C01791=1027.704,285.266,-126.131,170.638,46.717,159.004
C01792=1027.711,285.514,-126.162,170.643,46.715,159.005
C01793=1027.718,285.761,-126.193,170.647,46.714,159.005
C01794=1027.724,286.009,-126.225,170.651,46.713,159.005
C01795=1027.731,286.257,-126.256,170.655,46.712,159.005
C01796=1027.738,286.505,-126.288,170.660,46.711,159.006
C01797=1027.744,286.753,-126.319,170.664,46.710,159.006
C01798=1027.751,287.001,-126.351,170.668,46.709,159.006
C01799=1027.758,287.249,-126.382,170.673,46.708,159.006
C01800=1027.764,287.497,-126.414,170.678,46.706,159.007
C01801=1027.771,287.744,-126.446,170.682,46.705,159.007
C01802=1027.778,287.992,-126.478,170.686,46.704,159.007
C01803=1027.784,288.240,-126.509,170.690,46.703,159.008
C01804=1027.791,288.488,-126.541,170.695,46.702,159.008
C01805=1027.798,288.736,-126.572,170.699,46.701,159.008
C01806=1027.805,288.983,-126.604,170.703,46.700,159.008
C01807=1027.811,289.232,-126.636,170.708,46.699,159.009
C01808=1027.818,289.479,-126.668,170.712,46.698,159.009
C01809=1027.824,289.727,-126.699,170.716,46.697,159.009
C01810=1027.832,289.975,-126.732,170.720,46.696,159.010
C01811=1027.839,290.223,-126.763,170.725,46.695,159.010
C01812=1027.845,290.471,-126.795,170.730,46.694,159.010
C01813=1027.852,290.719,-126.827,170.734,46.693,159.011
C01814=1027.858,290.967,-126.859,170.739,46.692,159.011
C01815=1027.865,291.215,-126.890,170.743,46.691,159.011
C01816=1027.872,291.462,-126.922,170.747,46.690,159.011
C01817=1027.883,291.868,-126.974,170.754,46.689,159.012
C01818=1027.894,292.273,-127.027,170.761,46.687,159.012
C01819=1027.906,292.679,-127.079,170.769,46.685,159.013
C01820=1027.917,293.084,-127.132,170.776,46.684,159.014
C01821=1027.923,293.332,-127.163,170.781,46.683,159.014
C01822=1027.930,293.579,-127.196,170.785,46.682,159.014
C01823=1027.937,293.828,-127.228,170.789,46.681,159.015
C01824=1027.944,294.075,-127.260,170.794,46.680,159.015
C01825=1027.950,294.323,-127.293,170.798,46.679,159.015
C01826=1027.957,294.571,-127.324,170.803,46.679,159.016
C01827=1027.963,294.818,-127.357,170.807,46.678,159.016
C01828=1027.970,295.066,-127.390,170.812,46.677,159.016
C01829=1027.977,295.314,-127.422,170.816,46.676,159.017
C01830=1027.983,295.562,-127.454,170.821,46.675,159.017
C01831=1027.990,295.810,-127.487,170.826,46.675,159.018
C01832=1027.997,296.058,-127.519,170.830,46.674,159.018
C01833=1028.003,296.305,-127.552,170.834,46.673,159.018
C01834=1028.010,296.553,-127.585,170.838,46.672,159.019
C01835=1028.017,296.800,-127.617,170.844,46.671,159.019
C01836=1028.024,297.048,-127.650,170.848,46.671,159.019
C01837=1028.030,297.297,-127.682,170.852,46.670,159.020
C01838=1028.037,297.544,-127.714,170.857,46.669,159.020
C01839=1028.043,297.791,-127.747,170.861,46.668,159.020
C01840=1028.050,298.040,-127.780,170.866,46.668,159.021
C01841=1028.057,298.287,-127.812,170.871,46.667,159.021
C01842=1028.063,298.535,-127.845,170.875,46.666,159.022
C01843=1028.070,298.783,-127.878,170.879,46.666,159.022
C01844=1028.077,299.030,-127.910,170.885,46.665,159.023
C01845=1028.083,299.278,-127.943,170.889,46.665,159.023
C01846=1028.090,299.526,-127.976,170.893,46.663,159.023
C01847=1028.097,299.773,-128.008,170.898,46.663,159.024
C01848=1028.104,300.021,-128.041,170.903,46.662,159.024
C01849=1028.111,300.269,-128.074,170.908,46.661,159.024
C01850=1028.118,300.517,-128.106,170.912,46.661,159.025
C01851=1028.125,300.764,-128.140,170.917,46.660,159.025
C01852=1028.131,301.012,-128.173,170.922,46.659,159.026
C01853=1028.138,301.259,-128.205,170.926,46.659,159.026
C01854=1028.145,301.507,-128.238,170.930,46.658,159.026
C01855=1028.151,301.755,-128.271,170.936,46.657,159.027
C01856=1028.159,302.003,-128.303,170.940,46.657,159.027
C01857=1028.165,302.251,-128.336,170.945,46.656,159.028
C01858=1028.172,302.498,-128.370,170.950,46.656,159.028
C01859=1028.179,302.746,-128.403,170.954,46.655,159.029
C01860=1028.186,302.994,-128.435,170.959,46.654,159.029
C01861=1028.193,303.241,-128.468,170.963,46.654,159.029
C01862=1028.200,303.489,-128.502,170.969,46.653,159.030
C01863=1028.207,303.736,-128.534,170.973,46.652,159.030
C01864=1028.214,303.985,-128.567,170.978,46.652,159.031
C01865=1028.220,304.232,-128.601,170.983,46.651,159.031
C01866=1028.228,304.480,-128.633,170.987,46.651,159.032
C01867=1028.234,304.727,-128.666,170.992,46.650,159.032
C01868=1028.241,304.975,-128.700,170.996,46.649,159.032
C01869=1028.249,305.222,-128.732,171.002,46.648,159.033
C01870=1028.255,305.470,-128.765,171.006,46.648,159.033
C01871=1028.263,305.718,-128.799,171.011,46.647,159.034
C01872=1028.269,305.966,-128.831,171.016,46.647,159.034
C01873=1028.275,306.176,-128.860,171.020,46.646,159.035
C01874=1028.281,306.388,-128.888,171.024,46.646,159.035
C01875=1028.287,306.599,-128.917,171.029,46.646,159.036
C01876=1028.293,306.810,-128.944,171.032,46.645,159.036
C01877=1028.300,307.022,-128.973,171.036,46.644,159.036
C01878=1028.305,307.233,-129.001,171.040,46.644,159.037
C01879=1028.312,307.445,-129.030,171.045,46.644,159.037
C01880=1028.318,307.656,-129.057,171.049,46.643,159.037
C01881=1028.325,307.904,-129.091,171.053,46.643,159.038
C01882=1028.331,308.151,-129.124,171.059,46.642,159.038
C01883=1028.339,308.398,-129.157,171.063,46.642,159.039
C01884=1028.346,308.647,-129.190,171.068,46.641,159.039
C01885=1028.353,308.894,-129.224,171.073,46.641,159.040
C01886=1028.360,309.141,-129.258,171.078,46.640,159.040
C01887=1028.367,309.389,-129.290,171.083,46.640,159.041
C01888=1028.375,309.637,-129.324,171.088,46.639,159.041
C01889=1028.381,309.884,-129.357,171.092,46.639,159.042
C01890=1028.388,310.132,-129.390,171.098,46.638,159.042
C01891=1028.396,310.380,-129.424,171.102,46.638,159.043
C01892=1028.403,310.627,-129.458,171.107,46.637,159.043
C01893=1028.410,310.875,-129.490,171.112,46.637,159.044
C01894=1028.417,311.123,-129.524,171.117,46.636,159.044
C01895=1028.424,311.370,-129.558,171.122,46.636,159.045
C01896=1028.430,311.618,-129.592,171.127,46.636,159.045
C01897=1028.437,311.865,-129.626,171.132,46.635,159.046
C01898=1028.444,312.113,-129.660,171.137,46.635,159.046
C01899=1028.451,312.361,-129.693,171.142,46.635,159.047
C01900=1028.458,312.607,-129.728,171.147,46.635,159.047
C01901=1028.465,312.855,-129.762,171.151,46.634,159.048
C01902=1028.472,313.103,-129.796,171.157,46.634,159.049
C01903=1028.478,313.351,-129.830,171.161,46.634,159.049
C01904=1028.486,313.598,-129.864,171.167,46.634,159.050
C01905=1028.492,313.845,-129.898,171.171,46.633,159.050
C01906=1028.499,314.093,-129.932,171.177,46.633,159.051
C01907=1028.506,314.341,-129.966,171.181,46.633,159.051
C01908=1028.513,314.588,-130.001,171.187,46.633,159.052
C01909=1028.520,314.836,-130.035,171.192,46.633,159.052
C01910=1028.526,315.083,-130.068,171.197,46.632,159.053
C01911=1028.533,315.331,-130.103,171.202,46.633,159.054
C01912=1028.540,315.578,-130.137,171.207,46.632,159.054
C01913=1028.548,315.826,-130.171,171.213,46.632,159.055
C01914=1028.554,316.074,-130.205,171.217,46.632,159.055
C01915=1028.561,316.321,-130.239,171.223,46.631,159.056
C01916=1028.569,316.568,-130.274,171.227,46.631,159.056
C01917=1028.575,316.816,-130.308,171.233,46.631,159.057
C01918=1028.582,317.064,-130.342,171.237,46.631,159.057
C01919=1028.590,317.311,-130.377,171.243,46.631,159.058
C01920=1028.596,317.559,-130.411,171.248,46.631,159.059
C01921=1028.604,317.806,-130.446,171.253,46.630,159.059
C01922=1028.611,318.053,-130.479,171.258,46.630,159.060
C01923=1028.617,318.301,-130.513,171.263,46.630,159.060
C01924=1028.624,318.548,-130.548,171.269,46.630,159.061
C01925=1028.632,318.797,-130.583,171.273,46.630,159.062
C01926=1028.639,319.044,-130.617,171.279,46.630,159.062
C01927=1028.646,319.292,-130.651,171.284,46.630,159.063
C01928=1028.653,319.539,-130.686,171.289,46.630,159.063
C01929=1028.660,319.787,-130.720,171.294,46.629,159.064
C01930=1028.668,320.034,-130.755,171.300,46.629,159.065
C01931=1028.674,320.282,-130.789,171.304,46.629,159.065
C01932=1028.682,320.529,-130.824,171.310,46.629,159.066
C01933=1028.688,320.743,-130.854,171.315,46.629,159.066
C01934=1028.694,320.957,-130.884,171.319,46.629,159.067
C01935=1028.700,321.170,-130.913,171.324,46.629,159.068
C01936=1028.706,321.384,-130.943,171.328,46.629,159.068
C01937=1028.712,321.597,-130.973,171.333,46.629,159.069
C01938=1028.719,321.811,-131.003,171.337,46.629,159.069
C01939=1028.725,322.025,-131.033,171.342,46.629,159.070
C01940=1028.731,322.239,-131.063,171.346,46.629,159.070
C01941=1028.739,322.486,-131.097,171.352,46.629,159.071
C01942=1028.746,322.733,-131.132,171.356,46.629,159.071
C01943=1028.753,322.981,-131.166,171.362,46.629,159.072
C01944=1028.760,323.229,-131.201,171.368,46.629,159.073
C01945=1028.767,323.477,-131.236,171.373,46.629,159.073
C01946=1028.775,323.724,-131.271,171.378,46.629,159.074
C01947=1028.782,323.971,-131.305,171.384,46.629,159.075
C01948=1028.789,324.219,-131.340,171.389,46.629,159.075
C01949=1028.797,324.466,-131.375,171.394,46.629,159.076
C01950=1028.804,324.714,-131.410,171.399,46.629,159.077
C01951=1028.811,324.961,-131.445,171.405,46.629,159.077
C01952=1028.819,325.209,-131.479,171.411,46.629,159.078
C01953=1028.826,325.456,-131.515,171.415,46.629,159.079
C01954=1028.834,325.703,-131.549,171.421,46.629,159.079
C01955=1028.841,325.951,-131.585,171.427,46.629,159.080
C01956=1028.849,326.198,-131.619,171.433,46.629,159.081
C01957=1028.855,326.446,-131.654,171.437,46.629,159.081
C01958=1028.863,326.693,-131.689,171.443,46.629,159.082
C01959=1028.871,326.940,-131.724,171.448,46.629,159.083
C01960=1028.878,327.188,-131.759,171.454,46.629,159.083
C01961=1028.886,327.435,-131.794,171.459,46.630,159.084
C01962=1028.893,327.683,-131.829,171.465,46.630,159.085
C01963=1028.900,327.931,-131.864,171.470,46.630,159.085
C01964=1028.907,328.178,-131.899,171.476,46.630,159.086
C01965=1028.915,328.425,-131.935,171.481,46.630,159.087
C01966=1028.922,328.673,-131.970,171.486,46.630,159.087
C01967=1028.929,328.920,-132.005,171.492,46.631,159.088
C01968=1028.936,329.167,-132.041,171.498,46.631,159.089
C01969=1028.943,329.415,-132.077,171.503,46.632,159.090
C01970=1028.951,329.662,-132.111,171.509,46.632,159.090
C01971=1028.958,329.909,-132.148,171.515,46.632,159.091
C01972=1028.965,330.157,-132.183,171.520,46.632,159.092
C01973=1028.973,330.404,-132.219,171.526,46.632,159.093
C01974=1028.980,330.652,-132.254,171.531,46.633,159.093
C01975=1028.987,330.899,-132.290,171.537,46.633,159.094
C01976=1028.994,331.146,-132.325,171.542,46.633,159.095
C01977=1029.002,331.394,-132.361,171.548,46.634,159.096
C01978=1029.009,331.641,-132.396,171.554,46.633,159.096
C01979=1029.017,331.888,-132.432,171.559,46.634,159.097
C01980=1029.024,332.136,-132.468,171.565,46.635,159.098
C01981=1029.031,332.383,-132.504,171.570,46.635,159.099
C01982=1029.038,332.631,-132.539,171.576,46.635,159.100
C01983=1029.046,332.878,-132.575,171.582,46.636,159.100
C01984=1029.054,333.124,-132.610,171.588,46.636,159.101
C01985=1029.061,333.372,-132.646,171.593,46.636,159.102
C01986=1029.069,333.620,-132.682,171.599,46.637,159.103
C01987=1029.076,333.867,-132.718,171.604,46.637,159.103
C01988=1029.083,334.115,-132.753,171.610,46.637,159.104
C01989=1029.091,334.362,-132.790,171.616,46.638,159.105
C01990=1029.098,334.609,-132.825,171.622,46.638,159.106
C01991=1029.105,334.856,-132.862,171.627,46.639,159.106
C01992=1029.113,335.103,-132.898,171.633,46.639,159.107
C01993=1029.119,335.315,-132.929,171.638,46.640,159.108
C01994=1029.125,335.527,-132.959,171.643,46.640,159.109
C01995=1029.131,335.738,-132.991,171.648,46.641,159.109
C01996=1029.137,335.950,-133.022,171.653,46.641,159.110
C01997=1029.144,336.162,-133.052,171.658,46.642,159.111
C01998=1029.150,336.372,-133.084,171.662,46.642,159.111
C01999=1029.156,336.584,-133.114,171.668,46.642,159.112
C02000=1029.163,336.796,-133.145,171.673,46.642,159.113
C02001=1029.170,337.043,-133.182,171.679,46.643,159.114
C02002=1029.178,337.290,-133.218,171.685,46.643,159.115
C02003=1029.185,337.537,-133.254,171.690,46.644,159.115
C02004=1029.193,337.785,-133.290,171.696,46.645,159.116
C02005=1029.200,338.032,-133.326,171.701,46.645,159.117
C02006=1029.208,338.279,-133.362,171.707,46.646,159.118
C02007=1029.215,338.527,-133.399,171.713,46.646,159.119
C02008=1029.222,338.774,-133.435,171.719,46.647,159.120
C02009=1029.230,339.022,-133.472,171.725,46.648,159.121
C02010=1029.238,339.269,-133.509,171.731,46.648,159.121
C02011=1029.245,339.515,-133.544,171.737,46.649,159.122
C02012=1029.253,339.763,-133.581,171.743,46.649,159.123
C02013=1029.260,340.010,-133.617,171.749,46.650,159.124
C02014=1029.268,340.257,-133.654,171.755,46.650,159.125
C02015=1029.275,340.505,-133.691,171.761,46.651,159.126
C02016=1029.283,340.752,-133.727,171.767,46.652,159.127
C02017=1029.291,340.999,-133.764,171.773,46.653,159.128
C02018=1029.297,341.246,-133.800,171.779,46.653,159.128
C02019=1029.305,341.493,-133.837,171.785,46.654,159.129
C02020=1029.313,341.740,-133.873,171.791,46.655,159.130
C02021=1029.320,341.987,-133.911,171.797,46.655,159.131
C02022=1029.328,342.235,-133.947,171.803,46.656,159.132
C02023=1029.335,342.482,-133.985,171.809,46.657,159.133
C02024=1029.343,342.730,-134.021,171.815,46.657,159.134
C02025=1029.351,342.976,-134.058,171.822,46.658,159.135
C02026=1029.358,343.223,-134.095,171.827,46.659,159.136
C02027=1029.366,343.471,-134.132,171.834,46.660,159.137
C02028=1029.373,343.718,-134.169,171.840,46.661,159.138
C02029=1029.381,343.965,-134.206,171.846,46.662,159.139
C02030=1029.389,344.212,-134.242,171.852,46.662,159.139
C02031=1029.396,344.459,-134.280,171.858,46.663,159.140
C02032=1029.404,344.706,-134.317,171.864,46.664,159.141
C02033=1029.411,344.953,-134.354,171.870,46.665,159.142
C02034=1029.419,345.201,-134.390,171.876,46.665,159.143
C02035=1029.426,345.448,-134.428,171.882,46.666,159.144
C02036=1029.434,345.695,-134.465,171.889,46.668,159.145
C02037=1029.441,345.942,-134.502,171.895,46.668,159.146
C02038=1029.450,346.189,-134.540,171.901,46.669,159.147
C02039=1029.457,346.437,-134.577,171.908,46.670,159.148
C02040=1029.465,346.683,-134.614,171.914,46.671,159.149
C02041=1029.472,346.931,-134.652,171.920,46.672,159.150
C02042=1029.480,347.177,-134.689,171.926,46.673,159.151
C02043=1029.488,347.425,-134.726,171.932,46.673,159.152
C02044=1029.496,347.672,-134.763,171.939,46.674,159.153
C02045=1029.503,347.919,-134.801,171.945,46.675,159.154
C02046=1029.511,348.166,-134.838,171.951,46.677,159.155
C02047=1029.519,348.413,-134.875,171.958,46.677,159.156
C02048=1029.527,348.660,-134.912,171.964,46.678,159.157
C02049=1029.534,348.908,-134.950,171.970,46.679,159.158
C02050=1029.542,349.154,-134.989,171.977,46.680,159.159
C02051=1029.550,349.401,-135.025,171.983,46.681,159.160
C02052=1029.557,349.648,-135.063,171.989,46.682,159.161
C02053=1029.563,349.858,-135.095,171.995,46.683,159.162
C02054=1029.570,350.068,-135.127,172.000,46.684,159.163
C02055=1029.577,350.279,-135.160,172.006,46.685,159.164
C02056=1029.584,350.488,-135.191,172.011,46.686,159.165
C02057=1029.590,350.699,-135.224,172.016,46.687,159.165
C02058=1029.597,350.908,-135.255,172.023,46.688,159.166
C02059=1029.603,351.118,-135.288,172.027,46.689,159.167
C02060=1029.610,351.328,-135.320,172.034,46.690,159.168
C02061=1029.618,351.576,-135.358,172.040,46.691,159.169
C02062=1029.625,351.822,-135.396,172.046,46.692,159.170
C02063=1029.633,352.069,-135.433,172.052,46.693,159.171
C02064=1029.641,352.316,-135.471,172.059,46.694,159.172
C02065=1029.649,352.563,-135.509,172.066,46.695,159.173
C02066=1029.656,352.810,-135.547,172.072,46.696,159.174
C02067=1029.665,353.057,-135.585,172.079,46.698,159.176
C02068=1029.672,353.304,-135.623,172.085,46.699,159.177
C02069=1029.680,353.551,-135.661,172.092,46.700,159.178
C02070=1029.688,353.798,-135.699,172.098,46.701,159.179
C02071=1029.696,354.045,-135.737,172.105,46.702,159.180
C02072=1029.704,354.292,-135.775,172.112,46.703,159.181
C02073=1029.712,354.539,-135.814,172.118,46.704,159.182
C02074=1029.720,354.786,-135.851,172.125,46.706,159.183
C02075=1029.728,355.033,-135.890,172.131,46.707,159.184
C02076=1029.736,355.279,-135.927,172.138,46.708,159.185
C02077=1029.744,355.527,-135.966,172.145,46.710,159.187
C02078=1029.752,355.773,-136.004,172.151,46.711,159.188
C02079=1029.760,356.020,-136.043,172.159,46.712,159.189
C02080=1029.767,356.267,-136.081,172.165,46.713,159.190
C02081=1029.776,356.514,-136.120,172.171,46.715,159.191
C02082=1029.784,356.761,-136.158,172.179,46.716,159.192
C02083=1029.791,357.008,-136.197,172.185,46.717,159.193
C02084=1029.799,357.255,-136.235,172.191,46.718,159.194
C02085=1029.807,357.501,-136.273,172.199,46.720,159.196
C02086=1029.815,357.749,-136.312,172.206,46.721,159.197
C02087=1029.823,357.996,-136.351,172.213,46.722,159.198
C02088=1029.831,358.242,-136.389,172.219,46.724,159.199
C02089=1029.839,358.490,-136.427,172.226,46.726,159.200
C02090=1029.847,358.737,-136.466,172.233,46.726,159.202
C02091=1029.855,358.983,-136.505,172.240,46.728,159.203
C02092=1029.863,359.230,-136.544,172.247,46.730,159.204
C02093=1029.871,359.477,-136.582,172.254,46.731,159.205
C02094=1029.879,359.724,-136.621,172.260,46.732,159.206
C02095=1029.887,359.970,-136.660,172.268,46.734,159.208
C02096=1029.895,360.218,-136.698,172.274,46.735,159.209
C02097=1029.904,360.464,-136.738,172.282,46.737,159.210
C02098=1029.912,360.711,-136.776,172.288,46.738,159.211
C02099=1029.920,360.958,-136.815,172.296,46.740,159.212
C02100=1029.927,361.205,-136.855,172.302,46.741,159.214
C02101=1029.935,361.452,-136.893,172.310,46.743,159.215
C02102=1029.944,361.699,-136.932,172.316,46.745,159.216
C02103=1029.952,361.945,-136.972,172.323,46.746,159.217
C02104=1029.959,362.192,-137.011,172.330,46.748,159.219
C02105=1029.968,362.439,-137.050,172.337,46.749,159.220
C02106=1029.976,362.685,-137.089,172.344,46.751,159.221
C02107=1029.983,362.933,-137.129,172.351,46.752,159.222
C02108=1029.992,363.179,-137.168,172.359,46.754,159.224
C02109=1030.000,363.426,-137.207,172.365,46.756,159.225
C02110=1030.008,363.673,-137.247,172.373,46.757,159.226
C02111=1030.016,363.920,-137.286,172.380,46.759,159.228
C02112=1030.025,364.167,-137.325,172.387,46.760,159.229
C02113=1030.032,364.379,-137.359,172.394,46.762,159.230
C02114=1030.038,364.592,-137.393,172.400,46.763,159.231
C02115=1030.046,364.805,-137.428,172.405,46.765,159.232
C02116=1030.053,365.019,-137.461,172.412,46.766,159.233
C02117=1030.060,365.232,-137.495,172.418,46.768,159.234
C02118=1030.067,365.445,-137.529,172.425,46.769,159.236
C02119=1030.075,365.658,-137.564,172.431,46.770,159.237
C02120=1030.081,365.871,-137.598,172.437,46.772,159.238
C02121=1030.089,366.118,-137.637,172.444,46.774,159.239
C02122=1030.098,366.364,-137.677,172.452,46.776,159.241
C02123=1030.106,366.611,-137.717,172.458,46.777,159.242
C02124=1030.114,366.858,-137.756,172.466,46.779,159.243
C02125=1030.123,367.104,-137.795,172.474,46.781,159.245
C02126=1030.131,367.352,-137.835,172.481,46.783,159.246
C02127=1030.140,367.598,-137.876,172.488,46.784,159.247
C02128=1030.148,367.845,-137.915,172.496,46.786,159.249
C02129=1030.156,368.092,-137.955,172.503,46.788,159.250
C02130=1030.164,368.338,-137.994,172.510,46.790,159.251
C02131=1030.173,368.584,-138.034,172.518,46.792,159.253
C02132=1030.181,368.832,-138.074,172.525,46.794,159.254
C02133=1030.190,369.078,-138.114,172.533,46.796,159.256
C02134=1030.199,369.324,-138.154,172.541,46.798,159.257
C02135=1030.206,369.571,-138.194,172.548,46.800,159.258
C02136=1030.214,369.817,-138.234,172.555,46.801,159.260
C02137=1030.223,370.065,-138.274,172.563,46.803,159.261
C02138=1030.231,370.311,-138.315,172.571,46.805,159.263
C02139=1030.239,370.558,-138.355,172.578,46.807,159.264
C02140=1030.248,370.804,-138.395,172.585,46.809,159.265
C02141=1030.256,371.051,-138.436,172.593,46.811,159.267
C02142=1030.265,371.297,-138.475,172.601,46.813,159.268
C02143=1030.273,371.544,-138.516,172.608,46.815,159.270
C02144=1030.282,371.791,-138.557,172.616,46.817,159.271
C02145=1030.290,372.037,-138.597,172.624,46.819,159.273
C02146=1030.298,372.283,-138.637,172.632,46.821,159.274
C02147=1030.307,372.531,-138.678,172.639,46.823,159.276
C02148=1030.315,372.777,-138.718,172.646,46.825,159.277
C02149=1030.323,373.023,-138.758,172.654,46.827,159.279
C02150=1030.332,373.270,-138.799,172.662,46.829,159.280
C02151=1030.341,373.516,-138.839,172.670,46.832,159.282
C02152=1030.350,373.763,-138.880,172.678,46.834,159.283
C02153=1030.358,374.009,-138.921,172.686,46.836,159.285
C02154=1030.367,374.256,-138.961,172.694,46.838,159.286
C02155=1030.375,374.502,-139.002,172.701,46.841,159.288
C02156=1030.384,374.749,-139.043,172.709,46.843,159.289
C02157=1030.392,374.995,-139.083,172.717,46.844,159.291
C02158=1030.401,375.242,-139.124,172.724,46.846,159.292
C02159=1030.409,375.488,-139.165,172.733,46.849,159.294
C02160=1030.418,375.735,-139.205,172.741,46.851,159.295
C02161=1030.427,375.981,-139.246,172.749,46.853,159.297
C02162=1030.435,376.228,-139.287,172.757,46.855,159.298
C02163=1030.445,376.474,-139.328,172.765,46.858,159.300
C02164=1030.453,376.721,-139.368,172.773,46.860,159.301
C02165=1030.462,376.967,-139.410,172.781,46.862,159.303
C02166=1030.471,377.214,-139.451,172.789,46.864,159.305
C02167=1030.479,377.460,-139.491,172.797,46.867,159.306
C02168=1030.488,377.706,-139.533,172.805,46.869,159.308
C02169=1030.497,377.953,-139.574,172.813,46.871,159.309
C02170=1030.505,378.199,-139.615,172.821,46.874,159.311
C02171=1030.514,378.445,-139.657,172.829,46.876,159.313
C02172=1030.522,378.692,-139.698,172.837,46.878,159.314
C02173=1030.530,378.915,-139.735,172.844,46.881,159.316
C02174=1030.538,379.139,-139.773,172.852,46.883,159.317
C02175=1030.546,379.363,-139.811,172.859,46.885,159.319
C02176=1030.553,379.586,-139.848,172.867,46.887,159.320
C02177=1030.561,379.810,-139.886,172.874,46.890,159.322
C02178=1030.570,380.034,-139.924,172.882,46.892,159.323
C02179=1030.578,380.258,-139.961,172.889,46.894,159.325
C02180=1030.586,380.480,-139.999,172.897,46.896,159.326
C02181=1030.594,380.727,-140.040,172.905,46.899,159.328
C02182=1030.603,380.974,-140.082,172.913,46.901,159.330
C02183=1030.612,381.220,-140.124,172.921,46.904,159.331
C02184=1030.621,381.466,-140.165,172.930,46.906,159.333
C02185=1030.630,381.713,-140.207,172.938,46.909,159.334
C02186=1030.639,381.959,-140.249,172.947,46.911,159.336
C02187=1030.647,382.206,-140.291,172.955,46.914,159.338
C02188=1030.656,382.452,-140.333,172.963,46.916,159.340
C02189=1030.665,382.699,-140.375,172.972,46.919,159.341
C02190=1030.674,382.944,-140.417,172.980,46.922,159.343
C02191=1030.683,383.191,-140.459,172.989,46.924,159.345
C02192=1030.692,383.437,-140.500,172.997,46.926,159.346
C02193=1030.701,383.683,-140.542,173.006,46.929,159.348
C02194=1030.710,383.930,-140.584,173.014,46.932,159.350
C02195=1030.719,384.175,-140.626,173.023,46.934,159.352
C02196=1030.728,384.422,-140.668,173.032,46.937,159.354
C02197=1030.737,384.668,-140.710,173.040,46.940,159.355
C02198=1030.746,384.914,-140.752,173.048,46.943,159.357
C02199=1030.755,385.160,-140.794,173.058,46.945,159.359
C02200=1030.765,385.406,-140.836,173.066,46.948,159.361
C02201=1030.774,385.652,-140.878,173.074,46.950,159.362
C02202=1030.783,385.899,-140.921,173.084,46.953,159.364
C02203=1030.792,386.145,-140.962,173.092,46.956,159.366
C02204=1030.802,386.391,-141.005,173.101,46.959,159.368
C02205=1030.810,386.637,-141.047,173.110,46.962,159.370
C02206=1030.820,386.884,-141.089,173.118,46.964,159.371
C02207=1030.829,387.130,-141.132,173.128,46.967,159.373
C02208=1030.838,387.376,-141.174,173.136,46.970,159.375
C02209=1030.847,387.622,-141.217,173.145,46.973,159.377
C02210=1030.857,387.868,-141.259,173.154,46.976,159.379
C02211=1030.865,388.114,-141.302,173.163,46.979,159.381
C02212=1030.875,388.360,-141.345,173.172,46.981,159.383
C02213=1030.884,388.607,-141.388,173.181,46.985,159.384
C02214=1030.893,388.853,-141.431,173.189,46.988,159.386
C02215=1030.902,389.098,-141.473,173.199,46.990,159.388
C02216=1030.912,389.345,-141.516,173.207,46.993,159.390
C02217=1030.920,389.591,-141.559,173.217,46.996,159.392
C02218=1030.930,389.837,-141.601,173.225,46.999,159.394
C02219=1030.940,390.083,-141.644,173.235,47.002,159.396
C02220=1030.948,390.329,-141.687,173.243,47.005,159.398
C02221=1030.958,390.576,-141.730,173.253,47.008,159.400
C02222=1030.967,390.821,-141.774,173.262,47.011,159.402
C02223=1030.977,391.067,-141.817,173.271,47.014,159.404
C02224=1030.985,391.314,-141.860,173.281,47.017,159.406
C02225=1030.995,391.559,-141.903,173.289,47.020,159.408
C02226=1031.004,391.805,-141.946,173.299,47.023,159.409
C02227=1031.014,392.052,-141.989,173.308,47.027,159.412
C02228=1031.023,392.297,-142.032,173.317,47.029,159.413
C02229=1031.032,392.544,-142.075,173.327,47.033,159.416
C02230=1031.042,392.790,-142.119,173.336,47.036,159.417
C02231=1031.051,393.036,-142.162,173.345,47.039,159.420
C02232=1031.061,393.281,-142.206,173.355,47.042,159.421
C02233=1031.071,393.545,-142.252,173.365,47.046,159.424
C02234=1031.081,393.811,-142.299,173.375,47.049,159.426
C02235=1031.092,394.074,-142.345,173.385,47.052,159.428
C02236=1031.101,394.338,-142.392,173.395,47.056,159.430
C02237=1031.111,394.584,-142.437,173.405,47.060,159.432
C02238=1031.121,394.830,-142.480,173.414,47.062,159.434
C02239=1031.130,395.076,-142.524,173.424,47.066,159.436
C02240=1031.139,395.322,-142.567,173.433,47.069,159.439
C02241=1031.149,395.568,-142.611,173.443,47.072,159.441
C02242=1031.158,395.814,-142.655,173.453,47.076,159.443
C02243=1031.168,396.061,-142.699,173.462,47.079,159.445
C02244=1031.178,396.306,-142.743,173.471,47.083,159.447
C02245=1031.187,396.551,-142.787,173.481,47.086,159.449
C02246=1031.197,396.797,-142.831,173.491,47.089,159.451
C02247=1031.207,397.043,-142.875,173.501,47.093,159.454
C02248=1031.216,397.289,-142.919,173.511,47.096,159.456
C02249=1031.225,397.521,-142.960,173.520,47.099,159.457
C02250=1031.235,397.753,-143.002,173.529,47.103,159.460
C02251=1031.244,397.986,-143.044,173.538,47.106,159.462
C02252=1031.253,398.218,-143.085,173.548,47.109,159.464
C02253=1031.262,398.450,-143.127,173.557,47.112,159.466
C02254=1031.271,398.682,-143.169,173.566,47.116,159.468
C02255=1031.280,398.914,-143.210,173.576,47.119,159.470
C02256=1031.290,399.145,-143.253,173.585,47.122,159.472
C02257=1031.300,399.392,-143.297,173.595,47.126,159.474
C02258=1031.309,399.637,-143.342,173.605,47.130,159.476
C02259=1031.319,399.883,-143.386,173.615,47.133,159.479
C02260=1031.329,400.128,-143.430,173.625,47.137,159.481
C02261=1031.339,400.374,-143.475,173.635,47.140,159.483
C02262=1031.348,400.620,-143.519,173.646,47.144,159.486
C02263=1031.359,400.866,-143.564,173.655,47.147,159.488
C02264=1031.368,401.112,-143.609,173.666,47.151,159.490
C02265=1031.378,401.357,-143.654,173.676,47.155,159.492
C02266=1031.388,401.603,-143.698,173.686,47.159,159.495
C02267=1031.398,401.849,-143.744,173.697,47.162,159.497
C02268=1031.408,402.095,-143.789,173.707,47.166,159.499
C02269=1031.417,402.340,-143.833,173.717,47.170,159.502
C02270=1031.427,402.586,-143.878,173.728,47.174,159.504
C02271=1031.438,402.832,-143.923,173.738,47.178,159.506
C02272=1031.447,403.077,-143.968,173.748,47.182,159.509
C02273=1031.457,403.323,-144.013,173.759,47.185,159.511
C02274=1031.468,403.568,-144.059,173.769,47.189,159.513
C02275=1031.477,403.814,-144.104,173.779,47.193,159.516
C02276=1031.488,404.060,-144.149,173.790,47.197,159.518
C02277=1031.498,404.305,-144.194,173.800,47.201,159.521
C02278=1031.507,404.551,-144.239,173.811,47.204,159.523
C02279=1031.518,404.797,-144.284,173.822,47.209,159.525
C02280=1031.527,405.042,-144.331,173.832,47.212,159.528
C02281=1031.537,405.288,-144.376,173.843,47.216,159.530
C02282=1031.548,405.534,-144.422,173.854,47.220,159.533
C02283=1031.558,405.779,-144.467,173.864,47.224,159.535
C02284=1031.568,406.025,-144.512,173.875,47.228,159.538
C02285=1031.578,406.270,-144.558,173.886,47.232,159.540
C02286=1031.589,406.516,-144.603,173.896,47.236,159.542
C02287=1031.599,406.762,-144.649,173.908,47.240,159.545
C02288=1031.609,407.006,-144.695,173.918,47.245,159.548
C02289=1031.619,407.252,-144.741,173.929,47.248,159.550
C02290=1031.629,407.499,-144.786,173.940,47.252,159.553
C02291=1031.640,407.744,-144.832,173.951,47.256,159.555
C02292=1031.650,407.989,-144.878,173.962,47.261,159.558
C02293=1031.661,408.247,-144.926,173.973,47.265,159.560
C02294=1031.672,408.505,-144.974,173.985,47.269,159.563
C02295=1031.683,408.763,-145.023,173.997,47.273,159.566
C02296=1031.694,409.021,-145.071,174.009,47.278,159.568
C02297=1031.705,409.267,-145.117,174.019,47.282,159.571
C02298=1031.716,409.512,-145.163,174.031,47.286,159.574
C02299=1031.727,409.757,-145.209,174.042,47.290,159.576
C02300=1031.736,410.003,-145.256,174.053,47.295,159.579
C02301=1031.747,410.249,-145.302,174.065,47.299,159.581
C02302=1031.758,410.495,-145.348,174.076,47.303,159.584
C02303=1031.769,410.740,-145.394,174.087,47.308,159.587
C02304=1031.778,410.985,-145.441,174.098,47.312,159.589
C02305=1031.789,411.230,-145.487,174.110,47.317,159.592
C02306=1031.799,411.476,-145.534,174.121,47.321,159.595
C02307=1031.810,411.721,-145.580,174.133,47.326,159.598
C02308=1031.821,411.966,-145.627,174.144,47.329,159.600
C02309=1031.831,412.212,-145.673,174.156,47.334,159.603
C02310=1031.842,412.457,-145.720,174.167,47.339,159.606
C02311=1031.853,412.703,-145.768,174.179,47.343,159.608
C02312=1031.864,412.948,-145.814,174.190,47.347,159.611
C02313=1031.874,413.194,-145.861,174.202,47.352,159.614
C02314=1031.884,413.439,-145.907,174.214,47.356,159.617
C02315=1031.895,413.685,-145.955,174.226,47.361,159.619
C02316=1031.906,413.930,-146.002,174.238,47.366,159.622
C02317=1031.916,414.175,-146.049,174.249,47.370,159.625
C02318=1031.927,414.420,-146.095,174.261,47.375,159.628
C02319=1031.939,414.666,-146.142,174.272,47.379,159.631
C02320=1031.949,414.911,-146.190,174.284,47.384,159.633
C02321=1031.961,415.156,-146.237,174.296,47.388,159.636
C02322=1031.971,415.401,-146.285,174.308,47.393,159.639
C02323=1031.983,415.647,-146.332,174.320,47.398,159.642
C02324=1031.993,415.892,-146.379,174.333,47.402,159.645
C02325=1032.005,416.138,-146.427,174.345,47.407,159.648
C02326=1032.015,416.383,-146.474,174.357,47.412,159.651
C02327=1032.026,416.628,-146.521,174.369,47.417,159.654
C02328=1032.037,416.874,-146.569,174.381,47.421,159.657
C02329=1032.048,417.118,-146.617,174.394,47.426,159.660
C02330=1032.059,417.364,-146.664,174.405,47.431,159.662
C02331=1032.070,417.609,-146.712,174.419,47.436,159.665
C02332=1032.081,417.854,-146.760,174.431,47.441,159.668
C02333=1032.092,418.100,-146.808,174.443,47.446,159.671
C02334=1032.103,418.345,-146.855,174.455,47.451,159.675
C02335=1032.114,418.590,-146.903,174.468,47.456,159.678
C02336=1032.125,418.835,-146.952,174.481,47.460,159.681
C02337=1032.137,419.080,-146.999,174.493,47.465,159.684
C02338=1032.148,419.325,-147.047,174.505,47.470,159.687
C02339=1032.159,419.570,-147.096,174.518,47.475,159.690
C02340=1032.170,419.816,-147.144,174.531,47.480,159.693
C02341=1032.182,420.061,-147.192,174.544,47.485,159.696
C02342=1032.193,420.306,-147.240,174.556,47.490,159.699
C02343=1032.204,420.550,-147.289,174.569,47.495,159.702
C02344=1032.215,420.796,-147.337,174.582,47.500,159.705
C02345=1032.227,421.041,-147.385,174.594,47.506,159.708
C02346=1032.238,421.285,-147.434,174.608,47.510,159.711
C02347=1032.249,421.531,-147.482,174.621,47.516,159.715
C02348=1032.260,421.776,-147.530,174.634,47.521,159.718
C02349=1032.272,422.020,-147.579,174.647,47.526,159.721
C02350=1032.284,422.267,-147.627,174.659,47.531,159.724
C02351=1032.295,422.511,-147.676,174.673,47.536,159.727
C02352=1032.307,422.756,-147.725,174.686,47.541,159.731
C02353=1032.319,423.025,-147.778,174.700,47.547,159.734
C02354=1032.332,423.293,-147.831,174.715,47.552,159.738
C02355=1032.345,423.561,-147.885,174.729,47.559,159.741
C02356=1032.357,423.829,-147.938,174.744,47.564,159.745
C02357=1032.369,424.073,-147.987,174.757,47.570,159.748
C02358=1032.380,424.318,-148.036,174.771,47.575,159.751
C02359=1032.392,424.563,-148.085,174.784,47.580,159.755
C02360=1032.404,424.808,-148.136,174.798,47.586,159.758
C02361=1032.415,425.052,-148.185,174.812,47.591,159.762
C02362=1032.427,425.297,-148.234,174.825,47.596,159.765
C02363=1032.439,425.543,-148.283,174.839,47.602,159.768
C02364=1032.450,425.787,-148.332,174.852,47.607,159.772
C02365=1032.463,426.032,-148.382,174.866,47.613,159.775
C02366=1032.474,426.277,-148.431,174.879,47.618,159.778
C02367=1032.486,426.522,-148.481,174.893,47.624,159.782
C02368=1032.498,426.767,-148.530,174.908,47.629,159.785
C02369=1032.510,427.011,-148.580,174.922,47.635,159.789
C02370=1032.521,427.256,-148.629,174.936,47.640,159.792
C02371=1032.534,427.501,-148.679,174.950,47.646,159.796
C02372=1032.546,427.746,-148.730,174.964,47.652,159.799
C02373=1032.557,427.990,-148.780,174.977,47.657,159.803
C02374=1032.569,428.236,-148.829,174.992,47.664,159.806
C02375=1032.581,428.480,-148.879,175.006,47.669,159.810
C02376=1032.593,428.725,-148.929,175.021,47.675,159.814
C02377=1032.605,428.969,-148.979,175.035,47.680,159.817
C02378=1032.617,429.215,-149.030,175.049,47.686,159.821
C02379=1032.629,429.458,-149.080,175.063,47.692,159.824
C02380=1032.641,429.703,-149.130,175.078,47.697,159.828
C02381=1032.654,429.948,-149.180,175.092,47.704,159.832
C02382=1032.665,430.193,-149.231,175.107,47.709,159.835
C02383=1032.678,430.437,-149.282,175.121,47.715,159.839
C02384=1032.690,430.682,-149.332,175.136,47.721,159.843
C02385=1032.702,430.927,-149.382,175.151,47.727,159.846
C02386=1032.715,431.171,-149.433,175.165,47.733,159.850
C02387=1032.727,431.416,-149.484,175.180,47.739,159.854
C02388=1032.739,431.660,-149.534,175.194,47.745,159.857
C02389=1032.752,431.904,-149.585,175.210,47.751,159.861
C02390=1032.764,432.149,-149.635,175.225,47.756,159.865
C02391=1032.777,432.393,-149.686,175.239,47.763,159.869
C02392=1032.789,432.638,-149.738,175.255,47.769,159.873
C02393=1032.801,432.882,-149.788,175.270,47.775,159.877
C02394=1032.814,433.127,-149.838,175.285,47.781,159.880
C02395=1032.827,433.372,-149.890,175.300,47.787,159.884
C02396=1032.839,433.616,-149.940,175.316,47.793,159.888
C02397=1032.851,433.861,-149.992,175.331,47.799,159.892
C02398=1032.865,434.105,-150.044,175.347,47.805,159.896
C02399=1032.877,434.349,-150.095,175.362,47.811,159.900
C02400=1032.889,434.594,-150.146,175.378,47.817,159.904
C02401=1032.903,434.838,-150.197,175.392,47.824,159.908
C02402=1032.915,435.082,-150.249,175.408,47.830,159.912
C02403=1032.928,435.327,-150.300,175.424,47.836,159.916
C02404=1032.941,435.571,-150.352,175.439,47.843,159.920
C02405=1032.953,435.816,-150.404,175.455,47.849,159.924
C02406=1032.966,436.060,-150.455,175.472,47.855,159.928
C02407=1032.979,436.304,-150.508,175.488,47.862,159.932
C02408=1032.992,436.548,-150.559,175.503,47.868,159.936
C02409=1033.004,436.793,-150.611,175.519,47.874,159.940
C02410=1033.018,437.037,-150.663,175.535,47.881,159.944
C02411=1033.030,437.281,-150.715,175.551,47.887,159.948
C02412=1033.044,437.525,-150.767,175.568,47.894,159.952
C02413=1033.057,437.782,-150.822,175.585,47.900,159.957
C02414=1033.071,438.040,-150.877,175.601,47.908,159.961
C02415=1033.085,438.296,-150.932,175.619,47.915,159.966
C02416=1033.098,438.553,-150.987,175.636,47.921,159.970
C02417=1033.111,438.798,-151.039,175.653,47.928,159.974
C02418=1033.125,439.042,-151.091,175.669,47.934,159.978
C02419=1033.138,439.286,-151.144,175.686,47.941,159.983
C02420=1033.151,439.531,-151.196,175.702,47.948,159.987
C02421=1033.164,439.775,-151.249,175.719,47.954,159.991
C02422=1033.177,440.018,-151.303,175.735,47.961,159.996
C02423=1033.191,440.263,-151.355,175.753,47.968,160.000
C02424=1033.204,440.507,-151.408,175.770,47.975,160.004
C02425=1033.217,440.751,-151.461,175.786,47.982,160.009
C02426=1033.231,440.994,-151.514,175.803,47.988,160.013
C02427=1033.244,441.238,-151.567,175.821,47.995,160.018
C02428=1033.258,441.483,-151.620,175.838,48.002,160.022
C02429=1033.272,441.727,-151.673,175.855,48.009,160.027
C02430=1033.285,441.971,-151.726,175.871,48.015,160.031
C02431=1033.299,442.214,-151.779,175.889,48.022,160.036
C02432=1033.312,442.459,-151.832,175.906,48.029,160.040
C02433=1033.325,442.703,-151.886,175.924,48.037,160.045
C02434=1033.339,442.946,-151.939,175.941,48.044,160.049
C02435=1033.353,443.191,-151.992,175.959,48.050,160.054
C02436=1033.367,443.434,-152.046,175.977,48.057,160.058
C02437=1033.381,443.677,-152.100,175.995,48.064,160.063
C02438=1033.395,443.919,-152.152,176.012,48.071,160.068
C02439=1033.410,444.163,-152.204,176.030,48.078,160.072
C02440=1033.425,444.407,-152.257,176.049,48.085,160.077
C02441=1033.441,444.650,-152.308,176.066,48.092,160.081
C02442=1033.457,444.894,-152.359,176.085,48.098,160.086
C02443=1033.474,445.137,-152.411,176.103,48.105,160.091
C02444=1033.492,445.381,-152.461,176.120,48.111,160.095
C02445=1033.509,445.625,-152.511,176.138,48.117,160.099
C02446=1033.527,445.869,-152.561,176.157,48.124,160.104
C02447=1033.546,446.113,-152.609,176.176,48.130,160.109
C02448=1033.566,446.358,-152.659,176.195,48.136,160.113
C02449=1033.586,446.602,-152.707,176.213,48.142,160.117
C02450=1033.606,446.845,-152.754,176.232,48.148,160.122
C02451=1033.627,447.089,-152.802,176.251,48.153,160.126
C02452=1033.648,447.335,-152.849,176.270,48.160,160.131
C02453=1033.671,447.579,-152.895,176.289,48.165,160.135
C02454=1033.693,447.823,-152.942,176.308,48.171,160.140
C02455=1033.716,448.068,-152.988,176.327,48.177,160.144
C02456=1033.739,448.313,-153.033,176.346,48.182,160.149
C02457=1033.764,448.558,-153.078,176.365,48.187,160.153
C02458=1033.788,448.802,-153.123,176.385,48.192,160.158
C02459=1033.813,449.048,-153.167,176.404,48.198,160.162
C02460=1033.838,449.293,-153.210,176.424,48.203,160.166
C02461=1033.865,449.537,-153.253,176.444,48.208,160.171
C02462=1033.891,449.783,-153.295,176.463,48.213,160.175
C02463=1033.918,450.029,-153.338,176.483,48.218,160.180
C02464=1033.946,450.273,-153.380,176.503,48.223,160.184
C02465=1033.974,450.519,-153.422,176.523,48.228,160.188
C02466=1034.003,450.765,-153.463,176.544,48.232,160.193
C02467=1034.032,451.010,-153.503,176.564,48.237,160.197
C02468=1034.062,451.255,-153.543,176.583,48.242,160.201
C02469=1034.092,451.500,-153.583,176.604,48.246,160.206
C02470=1034.122,451.747,-153.623,176.625,48.250,160.210
C02471=1034.154,451.992,-153.662,176.645,48.255,160.214
C02472=1034.185,452.237,-153.700,176.666,48.259,160.219
C02473=1034.231,452.584,-153.754,176.695,48.266,160.225
C02474=1034.278,452.931,-153.806,176.725,48.271,160.231
C02475=1033.992,452.993,-154.134,176.728,48.338,160.252
C02476=1033.949,452.671,-154.086,176.701,48.333,160.247
C02477=1033.905,452.348,-154.036,176.673,48.328,160.241
C02478=1033.874,452.102,-153.998,176.652,48.323,160.237
C02479=1033.843,451.857,-153.960,176.632,48.319,160.232
C02480=1033.811,451.612,-153.920,176.611,48.315,160.228
C02481=1033.781,451.365,-153.881,176.591,48.310,160.224
C02482=1033.751,451.120,-153.841,176.570,48.306,160.219
C02483=1033.722,450.875,-153.800,176.550,48.301,160.215
C02484=1033.693,450.629,-153.760,176.530,48.297,160.211
C02485=1033.664,450.384,-153.719,176.510,48.292,160.206
C02486=1033.637,450.139,-153.677,176.490,48.287,160.202
C02487=1033.609,449.894,-153.634,176.470,48.283,160.198
C02488=1033.582,449.648,-153.592,176.450,48.278,160.193
C02489=1033.556,449.403,-153.550,176.430,48.273,160.189
C02490=1033.529,449.158,-153.506,176.410,48.268,160.184
C02491=1033.505,448.913,-153.462,176.391,48.262,160.180
C02492=1033.479,448.668,-153.418,176.371,48.257,160.175
C02493=1033.455,448.423,-153.373,176.352,48.252,160.171
C02494=1033.432,448.178,-153.328,176.333,48.247,160.167
C02495=1033.409,447.933,-153.283,176.313,48.241,160.162
C02496=1033.386,447.690,-153.236,176.294,48.236,160.158
C02497=1033.363,447.444,-153.190,176.275,48.231,160.153
C02498=1033.342,447.200,-153.143,176.256,48.224,160.149
C02499=1033.321,446.956,-153.096,176.237,48.219,160.144
C02500=1033.300,446.711,-153.048,176.218,48.213,160.140
C02501=1033.279,446.468,-153.001,176.200,48.207,160.135
C02502=1033.260,446.223,-152.952,176.180,48.202,160.131
C02503=1033.241,445.979,-152.903,176.162,48.195,160.126
C02504=1033.222,445.735,-152.854,176.144,48.189,160.122
C02505=1033.204,445.492,-152.804,176.125,48.183,160.117
C02506=1033.186,445.247,-152.754,176.107,48.177,160.113
C02507=1033.169,445.003,-152.703,176.089,48.170,160.108
C02508=1033.152,444.759,-152.652,176.070,48.164,160.104
C02509=1033.136,444.517,-152.601,176.053,48.157,160.099
C02510=1033.120,444.273,-152.550,176.034,48.151,160.095
C02511=1033.105,444.029,-152.496,176.016,48.144,160.090
C02512=1033.091,443.786,-152.444,175.998,48.137,160.085
C02513=1033.077,443.544,-152.391,175.981,48.130,160.081
C02514=1033.063,443.299,-152.337,175.963,48.123,160.076
C02515=1033.049,443.056,-152.285,175.946,48.116,160.072
C02516=1033.035,442.812,-152.230,175.928,48.109,160.067
C02517=1033.022,442.568,-152.177,175.910,48.103,160.063
C02518=1033.008,442.324,-152.124,175.892,48.096,160.058
C02519=1032.995,442.081,-152.071,175.875,48.089,160.053
C02520=1032.980,441.836,-152.018,175.857,48.082,160.049
C02521=1032.967,441.592,-151.964,175.841,48.076,160.045
C02522=1032.954,441.349,-151.911,175.824,48.069,160.040
C02523=1032.940,441.105,-151.859,175.806,48.062,160.036
C02524=1032.927,440.861,-151.805,175.789,48.056,160.031
C02525=1032.913,440.616,-151.752,175.772,48.049,160.027
C02526=1032.900,440.372,-151.700,175.756,48.042,160.023
C02527=1032.887,440.128,-151.647,175.738,48.035,160.018
C02528=1032.873,439.884,-151.594,175.721,48.029,160.014
C02529=1032.860,439.640,-151.542,175.705,48.022,160.009
C02530=1032.847,439.396,-151.488,175.688,48.016,160.005
C02531=1032.834,439.152,-151.437,175.671,48.009,160.001
C02532=1032.821,438.908,-151.384,175.655,48.002,159.997
C02533=1032.808,438.664,-151.332,175.638,47.996,159.992
C02534=1032.793,438.405,-151.276,175.620,47.989,159.988
C02535=1032.779,438.148,-151.221,175.603,47.983,159.984
C02536=1032.766,437.890,-151.165,175.586,47.976,159.979
C02537=1032.753,437.631,-151.111,175.569,47.969,159.975
C02538=1032.739,437.387,-151.059,175.553,47.962,159.970
C02539=1032.726,437.142,-151.006,175.537,47.956,159.966
C02540=1032.713,436.899,-150.955,175.520,47.950,159.962
C02541=1032.701,436.654,-150.902,175.504,47.943,159.958
C02542=1032.687,436.410,-150.850,175.489,47.937,159.954
C02543=1032.675,436.166,-150.798,175.473,47.930,159.950
C02544=1032.662,435.921,-150.747,175.457,47.924,159.946
C02545=1032.650,435.677,-150.695,175.440,47.918,159.942
C02546=1032.636,435.433,-150.643,175.425,47.912,159.938
C02547=1032.623,435.189,-150.592,175.409,47.906,159.934
C02548=1032.611,434.943,-150.541,175.394,47.900,159.930
C02549=1032.598,434.700,-150.489,175.378,47.893,159.926
C02550=1032.586,434.455,-150.438,175.362,47.887,159.922
C02551=1032.573,434.211,-150.386,175.347,47.881,159.918
C02552=1032.560,433.967,-150.335,175.331,47.875,159.914
C02553=1032.547,433.722,-150.283,175.317,47.869,159.910
C02554=1032.535,433.478,-150.232,175.301,47.863,159.906
C02555=1032.522,433.233,-150.182,175.286,47.857,159.902
C02556=1032.510,432.989,-150.131,175.270,47.851,159.899
C02557=1032.496,432.744,-150.080,175.255,47.845,159.895
C02558=1032.485,432.499,-150.029,175.240,47.840,159.891
C02559=1032.472,432.255,-149.978,175.225,47.833,159.887
C02560=1032.460,432.011,-149.927,175.210,47.827,159.883
C02561=1032.447,431.766,-149.877,175.195,47.822,159.880
C02562=1032.435,431.522,-149.826,175.180,47.816,159.876
C02563=1032.422,431.277,-149.776,175.165,47.810,159.872
C02564=1032.410,431.032,-149.725,175.151,47.804,159.868
C02565=1032.398,430.788,-149.674,175.135,47.798,159.865
C02566=1032.386,430.543,-149.624,175.121,47.792,159.861
C02567=1032.373,430.298,-149.574,175.106,47.786,159.857
C02568=1032.361,430.054,-149.523,175.092,47.781,159.854
C02569=1032.349,429.809,-149.472,175.077,47.775,159.850
C02570=1032.337,429.564,-149.422,175.063,47.769,159.846
C02571=1032.325,429.320,-149.372,175.048,47.764,159.843
C02572=1032.313,429.075,-149.322,175.033,47.758,159.839
C02573=1032.300,428.831,-149.272,175.020,47.752,159.836
C02574=1032.288,428.586,-149.221,175.005,47.747,159.832
C02575=1032.277,428.342,-149.171,174.991,47.741,159.828
C02576=1032.265,428.096,-149.122,174.977,47.735,159.825
C02577=1032.252,427.852,-149.072,174.963,47.730,159.821
C02578=1032.241,427.608,-149.022,174.949,47.724,159.818
C02579=1032.229,427.362,-148.971,174.934,47.719,159.814
C02580=1032.217,427.118,-148.922,174.920,47.713,159.811
C02581=1032.205,426.873,-148.872,174.906,47.707,159.807
C02582=1032.193,426.628,-148.822,174.892,47.702,159.804
C02583=1032.182,426.383,-148.773,174.878,47.697,159.800
C02584=1032.169,426.138,-148.723,174.865,47.691,159.797
C02585=1032.158,425.894,-148.674,174.851,47.686,159.794
C02586=1032.147,425.649,-148.625,174.837,47.681,159.790
C02587=1032.134,425.404,-148.575,174.823,47.675,159.787
C02588=1032.123,425.159,-148.526,174.809,47.670,159.783
C02589=1032.111,424.914,-148.476,174.796,47.665,159.780
C02590=1032.099,424.669,-148.427,174.782,47.659,159.777
C02591=1032.088,424.424,-148.378,174.769,47.654,159.774
C02592=1032.076,424.179,-148.329,174.755,47.648,159.770
C02593=1032.064,423.935,-148.281,174.742,47.643,159.767
C02594=1032.052,423.664,-148.226,174.727,47.638,159.763
C02595=1032.039,423.394,-148.172,174.712,47.632,159.760
C02596=1032.027,423.124,-148.118,174.698,47.626,159.756
C02597=1032.014,422.854,-148.064,174.683,47.620,159.752
C02598=1032.002,422.607,-148.015,174.669,47.615,159.749
C02599=1031.990,422.363,-147.967,174.657,47.610,159.746
C02600=1031.978,422.118,-147.918,174.644,47.605,159.743
C02601=1031.967,421.873,-147.870,174.630,47.600,159.740
C02602=1031.956,421.628,-147.821,174.618,47.595,159.736
C02603=1031.944,421.383,-147.773,174.604,47.590,159.733
C02604=1031.933,421.138,-147.725,174.591,47.585,159.730
C02605=1031.922,420.893,-147.676,174.579,47.580,159.727
C02606=1031.910,420.648,-147.627,174.565,47.575,159.724
C02607=1031.899,420.403,-147.580,174.553,47.570,159.721
C02608=1031.888,420.157,-147.531,174.540,47.565,159.718
C02609=1031.876,419.912,-147.482,174.527,47.560,159.715
C02610=1031.865,419.668,-147.435,174.514,47.555,159.711
C02611=1031.854,419.423,-147.387,174.502,47.550,159.708
C02612=1031.843,419.177,-147.338,174.489,47.545,159.705
C02613=1031.832,418.932,-147.290,174.476,47.541,159.702
C02614=1031.820,418.687,-147.242,174.464,47.536,159.699
C02615=1031.809,418.442,-147.194,174.452,47.531,159.696
C02616=1031.798,418.196,-147.147,174.439,47.526,159.693
C02617=1031.787,417.951,-147.099,174.427,47.521,159.690
C02618=1031.776,417.707,-147.051,174.414,47.516,159.687
C02619=1031.765,417.461,-147.003,174.401,47.512,159.684
C02620=1031.754,417.215,-146.955,174.389,47.507,159.681
C02621=1031.743,416.971,-146.908,174.377,47.502,159.678
C02622=1031.732,416.726,-146.860,174.365,47.498,159.676
C02623=1031.722,416.480,-146.813,174.353,47.493,159.672
C02624=1031.710,416.235,-146.766,174.340,47.488,159.670
C02625=1031.699,415.989,-146.717,174.328,47.483,159.667
C02626=1031.688,415.744,-146.671,174.316,47.479,159.664
C02627=1031.677,415.499,-146.624,174.304,47.474,159.661
C02628=1031.666,415.254,-146.576,174.292,47.470,159.658
C02629=1031.655,415.008,-146.529,174.280,47.465,159.655
C02630=1031.644,414.763,-146.482,174.268,47.461,159.652
C02631=1031.633,414.518,-146.435,174.256,47.456,159.650
C02632=1031.623,414.272,-146.387,174.244,47.452,159.647
C02633=1031.612,414.027,-146.341,174.233,47.447,159.644
C02634=1031.602,413.782,-146.293,174.221,47.443,159.641
C02635=1031.590,413.536,-146.246,174.209,47.438,159.638
C02636=1031.580,413.291,-146.199,174.197,47.434,159.636
C02637=1031.569,413.046,-146.153,174.185,47.429,159.633
C02638=1031.558,412.801,-146.106,174.173,47.425,159.630
C02639=1031.547,412.555,-146.058,174.162,47.421,159.627
C02640=1031.537,412.309,-146.013,174.151,47.416,159.625
C02641=1031.526,412.064,-145.965,174.139,47.412,159.622
C02642=1031.515,411.819,-145.919,174.127,47.408,159.619
C02643=1031.506,411.573,-145.872,174.115,47.403,159.616
C02644=1031.495,411.328,-145.826,174.104,47.399,159.614
C02645=1031.485,411.082,-145.779,174.093,47.395,159.611
C02646=1031.474,410.837,-145.732,174.081,47.390,159.608
C02647=1031.463,410.592,-145.687,174.070,47.386,159.606
C02648=1031.453,410.346,-145.639,174.058,47.382,159.603
C02649=1031.442,410.101,-145.593,174.047,47.377,159.600
C02650=1031.432,409.855,-145.548,174.036,47.373,159.598
C02651=1031.421,409.610,-145.502,174.024,47.369,159.595
C02652=1031.410,409.365,-145.455,174.014,47.365,159.593
C02653=1031.400,409.119,-145.409,174.002,47.361,159.590
C02654=1031.388,408.859,-145.360,173.990,47.356,159.587
C02655=1031.377,408.598,-145.311,173.979,47.352,159.585
C02656=1031.367,408.338,-145.263,173.967,47.348,159.582
C02657=1031.356,408.077,-145.215,173.955,47.344,159.579
C02658=1031.345,407.832,-145.169,173.944,47.340,159.577
C02659=1031.334,407.586,-145.123,173.933,47.335,159.574
C02660=1031.324,407.341,-145.077,173.922,47.332,159.572
C02661=1031.314,407.096,-145.031,173.912,47.328,159.569
C02662=1031.303,406.850,-144.986,173.900,47.324,159.567
C02663=1031.293,406.604,-144.940,173.890,47.320,159.564
C02664=1031.283,406.359,-144.894,173.878,47.316,159.562
C02665=1031.273,406.113,-144.848,173.868,47.312,159.559
C02666=1031.263,405.867,-144.803,173.857,47.308,159.557
C02667=1031.253,405.622,-144.758,173.846,47.304,159.554
C02668=1031.242,405.376,-144.712,173.836,47.300,159.552
C02669=1031.232,405.131,-144.667,173.825,47.297,159.549
C02670=1031.222,404.885,-144.621,173.814,47.292,159.547
C02671=1031.212,404.640,-144.576,173.804,47.288,159.544
C02672=1031.202,404.394,-144.531,173.793,47.285,159.542
C02673=1031.192,404.148,-144.485,173.782,47.281,159.540
C02674=1031.182,403.902,-144.440,173.772,47.277,159.537
C02675=1031.172,403.657,-144.395,173.761,47.273,159.535
C02676=1031.162,403.412,-144.349,173.751,47.269,159.532
C02677=1031.152,403.166,-144.304,173.740,47.266,159.530
C02678=1031.142,402.920,-144.259,173.730,47.262,159.528
C02679=1031.132,402.675,-144.214,173.720,47.258,159.525
C02680=1031.122,402.428,-144.169,173.709,47.255,159.523
C02681=1031.112,402.183,-144.124,173.699,47.251,159.521
C02682=1031.103,401.937,-144.080,173.688,47.247,159.518
C02683=1031.092,401.691,-144.034,173.678,47.244,159.516
C02684=1031.083,401.446,-143.990,173.668,47.240,159.514
C02685=1031.073,401.200,-143.945,173.658,47.236,159.512
C02686=1031.063,400.955,-143.900,173.647,47.233,159.509
C02687=1031.053,400.709,-143.856,173.637,47.229,159.507
C02688=1031.042,400.463,-143.810,173.627,47.226,159.505
C02689=1031.033,400.217,-143.766,173.617,47.222,159.502
C02690=1031.023,399.971,-143.722,173.607,47.219,159.500
C02691=1031.014,399.726,-143.677,173.597,47.215,159.498
C02692=1031.004,399.480,-143.633,173.587,47.211,159.496
C02693=1030.994,399.235,-143.588,173.577,47.208,159.494
C02694=1030.984,398.988,-143.544,173.567,47.204,159.491
C02695=1030.975,398.743,-143.499,173.557,47.201,159.489
C02696=1030.965,398.497,-143.455,173.547,47.197,159.487
C02697=1030.955,398.252,-143.411,173.537,47.194,159.485
C02698=1030.945,398.006,-143.367,173.527,47.191,159.483
C02699=1030.936,397.759,-143.323,173.517,47.188,159.480
C02700=1030.925,397.514,-143.279,173.507,47.184,159.478
C02701=1030.916,397.268,-143.235,173.497,47.181,159.476
C02702=1030.907,397.022,-143.190,173.487,47.177,159.474
C02703=1030.897,396.776,-143.147,173.477,47.174,159.472
C02704=1030.887,396.530,-143.103,173.468,47.170,159.470
C02705=1030.877,396.284,-143.058,173.459,47.167,159.468
C02706=1030.867,396.039,-143.014,173.449,47.164,159.465
C02707=1030.858,395.793,-142.971,173.439,47.161,159.463
C02708=1030.848,395.547,-142.927,173.429,47.158,159.461
C02709=1030.839,395.301,-142.883,173.419,47.155,159.459
C02710=1030.829,395.058,-142.841,173.411,47.151,159.457
C02711=1030.821,394.816,-142.797,173.401,47.148,159.455
C02712=1030.811,394.573,-142.754,173.391,47.145,159.453
C02713=1030.801,394.331,-142.711,173.382,47.141,159.451
C02714=1030.793,394.088,-142.668,173.373,47.139,159.449
C02715=1030.783,393.846,-142.625,173.363,47.135,159.447
C02716=1030.774,393.603,-142.582,173.354,47.132,159.445
C02717=1030.764,393.361,-142.539,173.345,47.129,159.443
C02718=1030.755,393.115,-142.496,173.335,47.126,159.441
C02719=1030.745,392.869,-142.452,173.326,47.123,159.439
C02720=1030.736,392.624,-142.410,173.317,47.120,159.437
C02721=1030.727,392.377,-142.366,173.307,47.117,159.435
C02722=1030.717,392.131,-142.323,173.298,47.114,159.433
C02723=1030.708,391.886,-142.279,173.289,47.111,159.431
C02724=1030.698,391.639,-142.236,173.279,47.108,159.429
C02725=1030.690,391.393,-142.193,173.270,47.105,159.427
C02726=1030.680,391.147,-142.150,173.261,47.102,159.425
C02727=1030.670,390.901,-142.107,173.251,47.099,159.423
C02728=1030.661,390.655,-142.064,173.243,47.096,159.421
C02729=1030.652,390.410,-142.021,173.233,47.093,159.419
C02730=1030.643,390.163,-141.977,173.224,47.090,159.417
C02731=1030.633,389.917,-141.935,173.215,47.087,159.415
C02732=1030.625,389.671,-141.892,173.206,47.084,159.414
C02733=1030.615,389.425,-141.849,173.197,47.081,159.412
C02734=1030.606,389.179,-141.807,173.188,47.078,159.410
C02735=1030.596,388.932,-141.764,173.179,47.076,159.408
C02736=1030.587,388.686,-141.721,173.170,47.073,159.406
C02737=1030.578,388.441,-141.679,173.161,47.070,159.404
C02738=1030.568,388.194,-141.636,173.152,47.067,159.402
C02739=1030.560,387.948,-141.593,173.143,47.064,159.400
C02740=1030.551,387.702,-141.550,173.134,47.061,159.398
C02741=1030.541,387.456,-141.507,173.125,47.059,159.397
C02742=1030.533,387.209,-141.465,173.117,47.056,159.395
C02743=1030.523,386.963,-141.423,173.107,47.053,159.393
C02744=1030.514,386.718,-141.380,173.098,47.050,159.391
C02745=1030.504,386.471,-141.338,173.089,47.048,159.389
C02746=1030.490,386.079,-141.271,173.076,47.044,159.386
C02747=1030.476,385.688,-141.203,173.062,47.039,159.384
C02748=1030.461,385.295,-141.136,173.048,47.035,159.381
C02749=1030.446,384.904,-141.070,173.034,47.031,159.378
C02750=1030.437,384.657,-141.027,173.025,47.028,159.376
C02751=1030.429,384.411,-140.986,173.016,47.025,159.374
C02752=1030.419,384.165,-140.943,173.008,47.023,159.373
C02753=1030.410,383.919,-140.901,173.000,47.020,159.371
C02754=1030.401,383.672,-140.860,172.991,47.018,159.369
C02755=1030.392,383.426,-140.817,172.982,47.015,159.367
C02756=1030.383,383.180,-140.776,172.974,47.013,159.366
C02757=1030.374,382.934,-140.734,172.965,47.010,159.364
C02758=1030.365,382.687,-140.692,172.957,47.008,159.362
C02759=1030.356,382.441,-140.650,172.949,47.006,159.361
C02760=1030.347,382.195,-140.609,172.940,47.002,159.359
C02761=1030.339,381.948,-140.567,172.932,47.000,159.357
C02762=1030.330,381.702,-140.525,172.923,46.998,159.355
C02763=1030.321,381.456,-140.484,172.914,46.995,159.354
C02764=1030.312,381.209,-140.442,172.906,46.993,159.352
C02765=1030.303,380.963,-140.400,172.898,46.990,159.350
C02766=1030.294,380.717,-140.359,172.890,46.988,159.349
C02767=1030.286,380.471,-140.317,172.881,46.986,159.347
C02768=1030.277,380.224,-140.275,172.873,46.983,159.345
C02769=1030.268,379.978,-140.234,172.865,46.981,159.344
C02770=1030.257,379.675,-140.183,172.855,46.978,159.342
C02771=1030.246,379.370,-140.132,172.844,46.975,159.340
C02772=1030.235,379.067,-140.080,172.834,46.972,159.338
C02773=1030.225,378.764,-140.030,172.824,46.969,159.336
C02774=1030.216,378.517,-139.989,172.816,46.967,159.334
C02775=1030.208,378.271,-139.947,172.808,46.965,159.332
C02776=1030.199,378.025,-139.906,172.800,46.962,159.331
C02777=1030.190,377.778,-139.865,172.792,46.960,159.329
C02778=1030.182,377.532,-139.823,172.784,46.958,159.328
C02779=1030.173,377.285,-139.782,172.775,46.955,159.326
C02780=1030.165,377.038,-139.741,172.768,46.953,159.324
C02781=1030.156,376.793,-139.701,172.759,46.951,159.323
C02782=1030.147,376.546,-139.660,172.752,46.949,159.321
C02783=1030.138,376.299,-139.619,172.743,46.947,159.320
C02784=1030.129,376.053,-139.578,172.735,46.945,159.318
C02785=1030.121,375.806,-139.537,172.728,46.943,159.317
C02786=1030.112,375.559,-139.496,172.719,46.940,159.315
C02787=1030.103,375.313,-139.456,172.712,46.938,159.314
C02788=1030.095,375.066,-139.415,172.704,46.936,159.312
C02789=1030.087,374.820,-139.374,172.696,46.934,159.311
C02790=1030.077,374.573,-139.334,172.688,46.932,159.309
C02791=1030.069,374.327,-139.293,172.680,46.930,159.308
C02792=1030.061,374.080,-139.252,172.672,46.928,159.306
C02793=1030.052,373.834,-139.212,172.664,46.926,159.305
C02794=1030.043,373.587,-139.171,172.656,46.924,159.303
C02795=1030.035,373.341,-139.130,172.648,46.922,159.302
C02796=1030.026,373.095,-139.090,172.641,46.920,159.300
C02797=1030.018,372.848,-139.049,172.633,46.918,159.299
C02798=1030.010,372.602,-139.009,172.625,46.915,159.297
C02799=1030.000,372.355,-138.968,172.617,46.914,159.296
C02800=1029.992,372.109,-138.928,172.610,46.912,159.294
C02801=1029.985,371.862,-138.888,172.602,46.910,159.293
C02802=1029.975,371.615,-138.847,172.594,46.908,159.291
C02803=1029.967,371.369,-138.807,172.587,46.906,159.290
C02804=1029.958,371.123,-138.767,172.579,46.904,159.288
C02805=1029.950,370.875,-138.726,172.572,46.902,159.287
C02806=1029.942,370.629,-138.686,172.564,46.900,159.286
C02807=1029.933,370.383,-138.646,172.556,46.898,159.284
C02808=1029.926,370.136,-138.606,172.549,46.896,159.283
C02809=1029.917,369.889,-138.565,172.541,46.895,159.281
C02810=1029.908,369.642,-138.525,172.533,46.893,159.280
C02811=1029.900,369.396,-138.485,172.526,46.891,159.278
C02812=1029.893,369.149,-138.445,172.519,46.889,159.277
C02813=1029.884,368.903,-138.405,172.511,46.887,159.276
C02814=1029.875,368.656,-138.365,172.503,46.885,159.274
C02815=1029.867,368.409,-138.325,172.496,46.884,159.273
C02816=1029.859,368.162,-138.286,172.489,46.882,159.272
C02817=1029.850,367.917,-138.246,172.481,46.880,159.270
C02818=1029.842,367.670,-138.207,172.473,46.878,159.269
C02819=1029.833,367.422,-138.166,172.467,46.877,159.268
C02820=1029.825,367.176,-138.127,172.459,46.875,159.266
C02821=1029.816,366.929,-138.088,172.451,46.873,159.265
C02822=1029.809,366.682,-138.048,172.445,46.872,159.264
C02823=1029.800,366.436,-138.008,172.437,46.870,159.262
C02824=1029.791,366.190,-137.968,172.430,46.868,159.261
C02825=1029.784,365.943,-137.928,172.423,46.866,159.259
C02826=1029.776,365.729,-137.895,172.416,46.865,159.258
C02827=1029.769,365.514,-137.860,172.410,46.863,159.257
C02828=1029.762,365.300,-137.826,172.404,46.862,159.256
C02829=1029.755,365.086,-137.792,172.397,46.861,159.255
C02830=1029.747,364.871,-137.758,172.391,46.860,159.254
C02831=1029.741,364.657,-137.724,172.384,46.858,159.253
C02832=1029.734,364.443,-137.689,172.378,46.857,159.252
C02833=1029.726,364.229,-137.655,172.371,46.855,159.250
C02834=1029.718,363.983,-137.615,172.365,46.854,159.249
C02835=1029.710,363.736,-137.576,172.357,46.852,159.248
C02836=1029.702,363.489,-137.537,172.351,46.851,159.247
C02837=1029.694,363.242,-137.498,172.343,46.849,159.245
C02838=1029.686,362.995,-137.458,172.336,46.847,159.244
C02839=1029.677,362.749,-137.419,172.329,46.846,159.243
C02840=1029.670,362.501,-137.380,172.322,46.844,159.241
C02841=1029.662,362.255,-137.341,172.315,46.843,159.240
C02842=1029.654,362.009,-137.301,172.307,46.841,159.239
C02843=1029.645,361.761,-137.263,172.301,46.840,159.238
C02844=1029.638,361.514,-137.223,172.293,46.838,159.236
C02845=1029.629,361.267,-137.184,172.286,46.837,159.235
C02846=1029.622,361.021,-137.145,172.279,46.836,159.234
C02847=1029.613,360.774,-137.107,172.273,46.834,159.233
C02848=1029.605,360.528,-137.067,172.265,46.833,159.232
C02849=1029.598,360.280,-137.028,172.259,46.831,159.230
C02850=1029.589,360.033,-136.989,172.252,46.829,159.229
C02851=1029.582,359.787,-136.951,172.245,46.829,159.228
C02852=1029.573,359.540,-136.912,172.238,46.827,159.227
C02853=1029.565,359.292,-136.873,172.231,46.826,159.226
C02854=1029.557,359.046,-136.834,172.224,46.824,159.224
C02855=1029.549,358.799,-136.796,172.217,46.823,159.223
C02856=1029.541,358.552,-136.757,172.210,46.821,159.222
C02857=1029.533,358.305,-136.719,172.203,46.821,159.221
C02858=1029.525,358.058,-136.680,172.197,46.819,159.220
C02859=1029.517,357.812,-136.641,172.189,46.818,159.218
C02860=1029.509,357.565,-136.602,172.183,46.817,159.217
C02861=1029.501,357.318,-136.565,172.176,46.815,159.216
C02862=1029.492,357.071,-136.526,172.169,46.814,159.215
C02863=1029.485,356.825,-136.488,172.162,46.812,159.214
C02864=1029.477,356.577,-136.449,172.155,46.812,159.213
C02865=1029.469,356.330,-136.411,172.149,46.810,159.212
C02866=1029.461,356.084,-136.372,172.142,46.809,159.211
C02867=1029.453,355.837,-136.334,172.135,46.808,159.209
C02868=1029.445,355.590,-136.296,172.129,46.806,159.208
C02869=1029.437,355.342,-136.258,172.122,46.805,159.207
C02870=1029.430,355.096,-136.219,172.115,46.804,159.206
C02871=1029.422,354.848,-136.181,172.109,46.803,159.205
C02872=1029.414,354.602,-136.143,172.102,46.802,159.204
C02873=1029.405,354.355,-136.105,172.095,46.801,159.203
C02874=1029.398,354.108,-136.067,172.089,46.800,159.202
C02875=1029.390,353.861,-136.028,172.082,46.798,159.201
C02876=1029.382,353.614,-135.990,172.075,46.797,159.199
C02877=1029.374,353.367,-135.953,172.069,46.796,159.198
C02878=1029.366,353.120,-135.915,172.063,46.795,159.197
C02879=1029.358,352.872,-135.877,172.055,46.794,159.196
C02880=1029.351,352.626,-135.839,172.049,46.793,159.195
C02881=1029.343,352.379,-135.802,172.042,46.792,159.194
C02882=1029.335,352.132,-135.763,172.035,46.791,159.193
C02883=1029.327,351.885,-135.725,172.029,46.790,159.192
C02884=1029.319,351.637,-135.687,172.023,46.789,159.191
C02885=1029.311,351.391,-135.650,172.017,46.788,159.190
C02886=1029.305,351.180,-135.617,172.011,46.787,159.189
C02887=1029.298,350.969,-135.585,172.005,46.786,159.188
C02888=1029.291,350.758,-135.552,171.999,46.785,159.187
C02889=1029.285,350.546,-135.521,171.994,46.784,159.186
C02890=1029.278,350.336,-135.488,171.988,46.783,159.185
C02891=1029.272,350.125,-135.456,171.983,46.783,159.185
C02892=1029.266,349.914,-135.424,171.977,46.782,159.184
C02893=1029.259,349.703,-135.392,171.972,46.781,159.183
C02894=1029.251,349.456,-135.354,171.966,46.780,159.182
C02895=1029.243,349.209,-135.316,171.960,46.779,159.181
C02896=1029.236,348.962,-135.279,171.953,46.778,159.180
C02897=1029.228,348.715,-135.242,171.946,46.777,159.179
C02898=1029.220,348.467,-135.204,171.940,46.776,159.178
C02899=1029.213,348.220,-135.166,171.934,46.775,159.177
C02900=1029.205,347.973,-135.129,171.928,46.775,159.176
C02901=1029.198,347.726,-135.092,171.921,46.774,159.175
C02902=1029.190,347.479,-135.055,171.915,46.773,159.174
C02903=1029.182,347.231,-135.017,171.909,46.772,159.173
C02904=1029.174,346.985,-134.980,171.902,46.771,159.172
C02905=1029.167,346.738,-134.942,171.896,46.770,159.171
C02906=1029.159,346.491,-134.905,171.890,46.770,159.170
C02907=1029.151,346.244,-134.868,171.883,46.769,159.169
C02908=1029.143,345.997,-134.831,171.877,46.768,159.168
C02909=1029.136,345.750,-134.793,171.871,46.767,159.167
C02910=1029.128,345.503,-134.757,171.865,46.766,159.166
C02911=1029.119,345.255,-134.719,171.859,46.766,159.165
C02912=1029.113,345.007,-134.682,171.852,46.764,159.164
C02913=1029.105,344.761,-134.646,171.846,46.764,159.163
C02914=1029.097,344.514,-134.608,171.840,46.763,159.162
C02915=1029.089,344.267,-134.571,171.834,46.762,159.161
C02916=1029.082,344.019,-134.534,171.827,46.762,159.160
C02917=1029.074,343.772,-134.497,171.821,46.761,159.159
C02918=1029.067,343.525,-134.460,171.815,46.761,159.159
C02919=1029.060,343.278,-134.424,171.809,46.759,159.157
C02920=1029.052,343.031,-134.387,171.803,46.759,159.157
C02921=1029.044,342.784,-134.349,171.797,46.759,159.156
C02922=1029.037,342.536,-134.313,171.791,46.757,159.155
C02923=1029.029,342.289,-134.275,171.785,46.757,159.154
C02924=1029.022,342.042,-134.239,171.779,46.756,159.153
C02925=1029.014,341.795,-134.203,171.773,46.756,159.152
C02926=1029.007,341.548,-134.166,171.767,46.755,159.151
C02927=1028.999,341.301,-134.129,171.761,46.754,159.150
C02928=1028.992,341.053,-134.093,171.755,46.754,159.150
C02929=1028.984,340.806,-134.055,171.749,46.753,159.149
C02930=1028.977,340.559,-134.019,171.743,46.752,159.148
C02931=1028.969,340.311,-133.983,171.737,46.752,159.147
C02932=1028.962,340.064,-133.945,171.731,46.751,159.146
C02933=1028.955,339.818,-133.909,171.725,46.751,159.145
C02934=1028.947,339.570,-133.873,171.719,46.750,159.144
C02935=1028.939,339.323,-133.837,171.713,46.750,159.143
C02936=1028.931,339.076,-133.800,171.707,46.749,159.143
C02937=1028.924,338.828,-133.764,171.701,46.749,159.142
C02938=1028.916,338.581,-133.727,171.695,46.748,159.141
C02939=1028.910,338.334,-133.691,171.689,46.748,159.140
C02940=1028.902,338.086,-133.655,171.683,46.747,159.139
C02941=1028.894,337.839,-133.619,171.677,46.747,159.138
C02942=1028.887,337.592,-133.582,171.671,46.746,159.137
C02943=1028.879,337.345,-133.545,171.665,46.746,159.137
C02944=1028.872,337.098,-133.510,171.660,46.745,159.136
C02945=1028.864,336.851,-133.473,171.654,46.745,159.135
C02946=1028.858,336.638,-133.443,171.649,46.745,159.134
C02947=1028.852,336.425,-133.412,171.643,46.745,159.134
C02948=1028.846,336.213,-133.380,171.638,46.744,159.133
C02949=1028.839,336.000,-133.349,171.634,46.744,159.132
C02950=1028.833,335.788,-133.318,171.629,46.743,159.131
C02951=1028.827,335.574,-133.287,171.623,46.743,159.131
C02952=1028.821,335.362,-133.256,171.619,46.743,159.130
C02953=1028.813,335.150,-133.225,171.614,46.742,159.129
C02954=1028.806,334.902,-133.188,171.608,46.742,159.129
C02955=1028.799,334.655,-133.153,171.602,46.742,159.128
C02956=1028.792,334.407,-133.117,171.596,46.741,159.127
C02957=1028.785,334.160,-133.081,171.590,46.741,159.126
C02958=1028.777,333.913,-133.045,171.585,46.740,159.125
C02959=1028.769,333.666,-133.009,171.580,46.740,159.125
C02960=1028.763,333.418,-132.974,171.574,46.740,159.124
C02961=1028.755,333.171,-132.937,171.568,46.740,159.123
C02962=1028.747,332.924,-132.902,171.562,46.739,159.122
C02963=1028.740,332.676,-132.867,171.556,46.739,159.122
C02964=1028.732,332.429,-132.830,171.551,46.739,159.121
C02965=1028.725,332.182,-132.795,171.545,46.738,159.120
C02966=1028.718,331.934,-132.759,171.539,46.738,159.119
C02967=1028.710,331.687,-132.723,171.534,46.738,159.119
C02968=1028.703,331.439,-132.688,171.528,46.738,159.118
C02969=1028.695,331.193,-132.652,171.523,46.737,159.117
C02970=1028.688,330.945,-132.617,171.517,46.737,159.116
C02971=1028.681,330.698,-132.581,171.511,46.737,159.116
C02972=1028.674,330.450,-132.546,171.505,46.737,159.115
C02973=1028.667,330.203,-132.511,171.501,46.737,159.114
C02974=1028.659,329.955,-132.474,171.495,46.736,159.113
C02975=1028.652,329.708,-132.439,171.489,46.736,159.113
C02976=1028.644,329.461,-132.404,171.483,46.736,159.112
C02977=1028.637,329.213,-132.368,171.478,46.736,159.111
C02978=1028.630,328.966,-132.333,171.472,46.736,159.111
C02979=1028.623,328.718,-132.297,171.467,46.735,159.110
C02980=1028.616,328.471,-132.262,171.461,46.735,159.109
C02981=1028.609,328.224,-132.227,171.456,46.735,159.108
C02982=1028.601,327.977,-132.191,171.450,46.735,159.108
C02983=1028.594,327.729,-132.156,171.445,46.735,159.107
C02984=1028.587,327.482,-132.121,171.439,46.735,159.106
C02985=1028.579,327.234,-132.086,171.434,46.735,159.106
C02986=1028.572,326.987,-132.051,171.428,46.735,159.105
C02987=1028.564,326.739,-132.016,171.423,46.735,159.104
C02988=1028.557,326.492,-131.981,171.417,46.735,159.104
C02989=1028.550,326.245,-131.946,171.412,46.734,159.103
C02990=1028.542,325.997,-131.911,171.406,46.734,159.102
C02991=1028.535,325.749,-131.876,171.401,46.735,159.102
C02992=1028.528,325.502,-131.842,171.395,46.735,159.101
C02993=1028.520,325.254,-131.806,171.389,46.735,159.100
C02994=1028.513,325.007,-131.772,171.385,46.735,159.100
C02995=1028.505,324.760,-131.737,171.379,46.735,159.099
C02996=1028.498,324.511,-131.702,171.374,46.735,159.098
C02997=1028.491,324.264,-131.668,171.368,46.735,159.098
C02998=1028.484,324.017,-131.633,171.364,46.735,159.097
C02999=1028.476,323.770,-131.598,171.358,46.735,159.097
C03000=1028.468,323.522,-131.563,171.352,46.736,159.096
C03001=1028.461,323.275,-131.528,171.347,46.736,159.095
C03002=1028.454,323.027,-131.494,171.342,46.735,159.095
C03003=1028.447,322.780,-131.459,171.336,46.736,159.094
C03004=1028.440,322.533,-131.425,171.331,46.736,159.093
C03005=1028.432,322.284,-131.390,171.325,46.736,159.093
C03006=1028.426,322.070,-131.360,171.321,46.736,159.092
C03007=1028.420,321.855,-131.329,171.316,46.736,159.092
C03008=1028.414,321.640,-131.300,171.312,46.736,159.091
C03009=1028.408,321.426,-131.270,171.307,46.736,159.090
C03010=1028.402,321.210,-131.240,171.303,46.736,159.090
C03011=1028.395,320.995,-131.210,171.298,46.737,159.089
C03012=1028.389,320.781,-131.180,171.294,46.736,159.089
C03013=1028.383,320.566,-131.150,171.289,46.737,159.088
C03014=1028.375,320.319,-131.115,171.284,46.737,159.088
C03015=1028.369,320.071,-131.081,171.278,46.737,159.087
C03016=1028.361,319.824,-131.046,171.273,46.737,159.086
C03017=1028.354,319.576,-131.013,171.268,46.738,159.086
C03018=1028.347,319.329,-130.977,171.262,46.738,159.085
C03019=1028.340,319.081,-130.944,171.258,46.737,159.085
C03020=1028.332,318.834,-130.909,171.252,46.738,159.084
C03021=1028.326,318.586,-130.875,171.247,46.738,159.084
C03022=1028.318,318.339,-130.840,171.242,46.738,159.083
C03023=1028.312,318.091,-130.806,171.237,46.739,159.082
C03024=1028.305,317.843,-130.772,171.231,46.739,159.082
C03025=1028.297,317.596,-130.737,171.227,46.739,159.081
C03026=1028.291,317.348,-130.703,171.221,46.739,159.081
C03027=1028.283,317.101,-130.668,171.216,46.740,159.080
C03028=1028.276,316.854,-130.635,171.211,46.740,159.080
C03029=1028.270,316.606,-130.600,171.206,46.740,159.079
C03030=1028.262,316.359,-130.566,171.201,46.740,159.078
C03031=1028.255,316.111,-130.532,171.196,46.741,159.078
C03032=1028.248,315.863,-130.497,171.190,46.741,159.077
C03033=1028.242,315.616,-130.464,171.186,46.741,159.077
C03034=1028.234,315.369,-130.429,171.180,46.741,159.076
C03035=1028.228,315.121,-130.395,171.176,46.742,159.076
C03036=1028.221,314.873,-130.361,171.170,46.742,159.075
C03037=1028.214,314.625,-130.327,171.165,46.742,159.074
C03038=1028.207,314.378,-130.293,171.160,46.742,159.074
C03039=1028.200,314.131,-130.258,171.155,46.743,159.073
C03040=1028.194,313.883,-130.224,171.150,46.743,159.073
C03041=1028.186,313.636,-130.190,171.145,46.744,159.072
C03042=1028.179,313.388,-130.157,171.140,46.744,159.072
C03043=1028.173,313.140,-130.122,171.135,46.744,159.071
C03044=1028.166,312.893,-130.089,171.130,46.744,159.071
C03045=1028.159,312.645,-130.055,171.125,46.745,159.070
C03046=1028.153,312.397,-130.020,171.120,46.745,159.070
C03047=1028.145,312.150,-129.987,171.115,46.746,159.069
C03048=1028.139,311.903,-129.953,171.110,46.746,159.069
C03049=1028.132,311.655,-129.919,171.105,46.746,159.068
C03050=1028.125,311.407,-129.885,171.100,46.747,159.068
C03051=1028.119,311.160,-129.851,171.095,46.747,159.067
C03052=1028.111,310.912,-129.818,171.090,46.747,159.066
C03053=1028.104,310.665,-129.784,171.086,46.748,159.066
C03054=1028.097,310.417,-129.750,171.080,46.749,159.066
C03055=1028.090,310.170,-129.717,171.076,46.749,159.065
C03056=1028.083,309.922,-129.684,171.071,46.750,159.065
C03057=1028.075,309.674,-129.650,171.065,46.750,159.064
C03058=1028.068,309.427,-129.616,171.061,46.750,159.064
C03059=1028.061,309.179,-129.584,171.055,46.751,159.063
C03060=1028.054,308.932,-129.550,171.051,46.751,159.063
C03061=1028.047,308.683,-129.517,171.046,46.752,159.062
C03062=1028.041,308.436,-129.484,171.041,46.753,159.062
C03063=1028.033,308.189,-129.451,171.036,46.753,159.061
C03064=1028.026,307.941,-129.417,171.031,46.754,159.061
C03065=1028.019,307.694,-129.384,171.027,46.755,159.060
C03066=1028.012,307.481,-129.356,171.022,46.756,159.060
C03067=1028.007,307.269,-129.327,171.018,46.756,159.060
C03068=1028.001,307.056,-129.299,171.014,46.756,159.059
C03069=1027.995,306.844,-129.271,171.009,46.757,159.059
C03070=1027.989,306.632,-129.243,171.005,46.758,159.059
C03071=1027.983,306.419,-129.214,171.002,46.758,159.058
C03072=1027.976,306.207,-129.186,170.997,46.759,159.058
C03073=1027.971,305.994,-129.157,170.993,46.759,159.057
C03074=1027.963,305.748,-129.124,170.988,46.760,159.057
C03075=1027.956,305.499,-129.091,170.983,46.760,159.056
C03076=1027.950,305.252,-129.058,170.978,46.761,159.056
C03077=1027.942,305.004,-129.025,170.974,46.762,159.056
C03078=1027.935,304.756,-128.992,170.969,46.763,159.055
C03079=1027.929,304.508,-128.959,170.964,46.763,159.055
C03080=1027.922,304.261,-128.925,170.959,46.764,159.054
C03081=1027.915,304.014,-128.893,170.955,46.765,159.054
C03082=1027.908,303.765,-128.860,170.950,46.766,159.053
C03083=1027.901,303.518,-128.826,170.945,46.766,159.053
C03084=1027.894,303.270,-128.794,170.940,46.767,159.053
C03085=1027.887,303.023,-128.761,170.936,46.767,159.052
C03086=1027.881,302.774,-128.728,170.931,46.768,159.052
C03087=1027.873,302.527,-128.696,170.926,46.769,159.051
C03088=1027.866,302.279,-128.662,170.922,46.769,159.051
C03089=1027.860,302.032,-128.629,170.917,46.770,159.050
C03090=1027.852,301.784,-128.597,170.913,46.771,159.050
C03091=1027.846,301.536,-128.564,170.907,46.772,159.050
C03092=1027.840,301.289,-128.531,170.903,46.772,159.049
C03093=1027.832,301.041,-128.499,170.898,46.774,159.049
C03094=1027.826,300.794,-128.465,170.894,46.774,159.049
C03095=1027.819,300.545,-128.432,170.888,46.775,159.048
C03096=1027.812,300.298,-128.400,170.884,46.776,159.048
C03097=1027.805,300.051,-128.367,170.880,46.776,159.047
C03098=1027.798,299.802,-128.334,170.874,46.777,159.047
C03099=1027.791,299.555,-128.302,170.870,46.778,159.047
C03100=1027.785,299.307,-128.269,170.865,46.779,159.046
C03101=1027.778,299.059,-128.236,170.861,46.780,159.046
C03102=1027.771,298.812,-128.204,170.857,46.780,159.045
C03103=1027.765,298.564,-128.171,170.851,46.781,159.045
C03104=1027.758,298.316,-128.138,170.847,46.782,159.045
C03105=1027.751,298.069,-128.106,170.842,46.783,159.044
C03106=1027.745,297.821,-128.073,170.838,46.784,159.044
C03107=1027.738,297.573,-128.040,170.834,46.784,159.043
C03108=1027.731,297.325,-128.009,170.829,46.786,159.043
C03109=1027.725,297.077,-127.976,170.824,46.786,159.043
C03110=1027.718,296.830,-127.943,170.820,46.787,159.042
C03111=1027.711,296.582,-127.911,170.815,46.788,159.042
C03112=1027.705,296.334,-127.878,170.811,46.789,159.042
C03113=1027.698,296.087,-127.845,170.806,46.789,159.041
C03114=1027.691,295.839,-127.813,170.801,46.791,159.041
C03115=1027.685,295.590,-127.781,170.797,46.791,159.041
C03116=1027.678,295.343,-127.748,170.792,46.792,159.040
C03117=1027.671,295.095,-127.716,170.788,46.793,159.040
C03118=1027.665,294.848,-127.683,170.784,46.794,159.040
C03119=1027.659,294.600,-127.651,170.778,46.795,159.039
C03120=1027.651,294.352,-127.619,170.774,46.796,159.039
C03121=1027.645,294.104,-127.586,170.770,46.797,159.039
C03122=1027.638,293.856,-127.555,170.765,46.797,159.038
C03123=1027.631,293.609,-127.522,170.761,46.798,159.038
C03124=1027.625,293.361,-127.490,170.757,46.800,159.038
C03125=1027.618,293.113,-127.458,170.752,46.800,159.037
C03126=1027.607,292.705,-127.405,170.744,46.802,159.037
C03127=1027.596,292.298,-127.352,170.737,46.804,159.036
C03128=1027.584,291.890,-127.300,170.730,46.805,159.036
C03129=1027.573,291.482,-127.248,170.723,46.807,159.035
C03130=1027.566,291.235,-127.215,170.718,46.808,159.035
C03131=1027.560,290.987,-127.184,170.714,46.809,159.034
C03132=1027.554,290.739,-127.152,170.710,46.811,159.034
C03133=1027.547,290.492,-127.120,170.705,46.812,159.034
C03134=1027.540,290.244,-127.088,170.701,46.813,159.034
C03135=1027.533,289.996,-127.057,170.696,46.813,159.033
C03136=1027.526,289.749,-127.025,170.691,46.815,159.033
C03137=1027.519,289.500,-126.993,170.687,46.816,159.033
C03138=1027.513,289.252,-126.961,170.683,46.817,159.032
C03139=1027.506,289.004,-126.929,170.678,46.818,159.032
C03140=1027.499,288.757,-126.897,170.674,46.819,159.032
C03141=1027.492,288.509,-126.866,170.670,46.820,159.032
C03142=1027.486,288.261,-126.835,170.665,46.822,159.031
C03143=1027.479,288.013,-126.803,170.661,46.823,159.031
C03144=1027.472,287.766,-126.771,170.657,46.824,159.031
C03145=1027.466,287.517,-126.739,170.652,46.825,159.030
C03146=1027.459,287.269,-126.708,170.648,46.826,159.030
C03147=1027.452,287.022,-126.676,170.644,46.827,159.030
C03148=1027.446,286.774,-126.645,170.639,46.829,159.030
C03149=1027.439,286.526,-126.613,170.635,46.830,159.029
C03150=1027.432,286.278,-126.582,170.631,46.831,159.029
C03151=1027.426,286.030,-126.550,170.627,46.832,159.029
C03152=1027.419,285.782,-126.519,170.622,46.834,159.029
C03153=1027.412,285.534,-126.488,170.618,46.835,159.028
C03154=1027.405,285.286,-126.456,170.614,46.836,159.028
C03155=1027.399,285.038,-126.425,170.609,46.837,159.028
C03156=1027.392,284.790,-126.393,170.605,46.838,159.028
C03157=1027.385,284.543,-126.362,170.601,46.839,159.027
C03158=1027.378,284.295,-126.330,170.596,46.841,159.027
C03159=1027.371,284.047,-126.300,170.592,46.842,159.027
C03160=1027.365,283.799,-126.269,170.588,46.843,159.027
C03161=1027.358,283.551,-126.237,170.584,46.845,159.026
C03162=1027.351,283.303,-126.206,170.579,46.847,159.026
C03163=1027.344,283.055,-126.175,170.575,46.848,159.026
C03164=1027.338,282.807,-126.143,170.571,46.849,159.026
C03165=1027.331,282.559,-126.112,170.566,46.850,159.025
C03166=1027.325,282.310,-126.081,170.562,46.852,159.025
C03167=1027.317,282.063,-126.050,170.558,46.853,159.025
C03168=1027.310,281.815,-126.019,170.554,46.854,159.025
C03169=1027.304,281.568,-125.988,170.550,46.856,159.025
C03170=1027.298,281.319,-125.957,170.545,46.857,159.024
C03171=1027.291,281.071,-125.925,170.541,46.858,159.024
C03172=1027.284,280.823,-125.894,170.537,46.860,159.024
C03173=1027.278,280.575,-125.863,170.533,46.861,159.024
C03174=1027.271,280.327,-125.832,170.529,46.862,159.023
C03175=1027.264,280.079,-125.801,170.525,46.864,159.023
C03176=1027.258,279.832,-125.771,170.521,46.865,159.023
C03177=1027.251,279.584,-125.739,170.516,46.866,159.023
C03178=1027.244,279.336,-125.708,170.512,46.868,159.023
C03179=1027.238,279.087,-125.677,170.508,46.869,159.022
C03180=1027.231,278.839,-125.646,170.504,46.871,159.022
C03181=1027.225,278.592,-125.615,170.499,46.872,159.022
C03182=1027.214,278.197,-125.566,170.493,46.874,159.022
C03183=1027.204,277.801,-125.517,170.486,46.876,159.021
C03184=1027.193,277.406,-125.467,170.480,46.879,159.021
C03185=1027.183,277.011,-125.418,170.473,46.881,159.021
C03186=1027.176,276.762,-125.388,170.469,46.882,159.021
C03187=1027.169,276.514,-125.357,170.465,46.884,159.020
C03188=1027.163,276.266,-125.326,170.461,46.886,159.020
C03189=1027.156,276.018,-125.296,170.456,46.887,159.020
C03190=1027.149,275.771,-125.265,170.453,46.889,159.020
C03191=1027.142,275.522,-125.235,170.448,46.890,159.020
C03192=1027.136,275.274,-125.204,170.445,46.891,159.020
C03193=1027.130,275.027,-125.173,170.441,46.893,159.020
C03194=1027.123,274.778,-125.143,170.436,46.895,159.019
C03195=1027.116,274.530,-125.112,170.432,46.896,159.019
C03196=1027.109,274.282,-125.081,170.428,46.897,159.019
C03197=1027.103,274.034,-125.051,170.424,46.899,159.019
C03198=1027.096,273.786,-125.020,170.420,46.901,159.019
C03199=1027.089,273.538,-124.990,170.416,46.902,159.018
C03200=1027.083,273.291,-124.959,170.412,46.904,159.018
C03201=1027.076,273.042,-124.929,170.408,46.905,159.018
C03202=1027.070,272.794,-124.898,170.404,46.907,159.018
C03203=1027.063,272.546,-124.868,170.399,46.909,159.018
C03204=1027.057,272.298,-124.838,170.396,46.910,159.018
C03205=1027.049,272.050,-124.808,170.392,46.912,159.018
C03206=1027.044,271.802,-124.777,170.388,46.913,159.017
C03207=1027.037,271.554,-124.746,170.384,46.915,159.017
C03208=1027.030,271.306,-124.716,170.379,46.917,159.017
C03209=1027.024,271.058,-124.685,170.376,46.918,159.017
C03210=1027.017,270.810,-124.655,170.372,46.919,159.017
C03211=1027.011,270.562,-124.625,170.368,46.921,159.017
C03212=1027.004,270.314,-124.595,170.364,46.923,159.017
C03213=1026.997,270.065,-124.564,170.360,46.925,159.017
C03214=1026.991,269.817,-124.534,170.356,46.927,159.016
C03215=1026.984,269.569,-124.504,170.352,46.928,159.016
C03216=1026.978,269.321,-124.474,170.348,46.929,159.016
C03217=1026.971,269.073,-124.444,170.344,46.931,159.016
C03218=1026.964,268.825,-124.413,170.340,46.933,159.016
C03219=1026.958,268.577,-124.384,170.336,46.935,159.016
C03220=1026.951,268.328,-124.354,170.332,46.937,159.016
C03221=1026.944,268.081,-124.324,170.328,46.938,159.016
C03222=1026.938,267.832,-124.293,170.324,46.940,159.015
C03223=1026.931,267.585,-124.263,170.321,46.942,159.015
C03224=1026.924,267.337,-124.233,170.317,46.943,159.015
C03225=1026.918,267.088,-124.203,170.312,46.945,159.015
C03226=1026.912,266.840,-124.174,170.308,46.947,159.015
C03227=1026.904,266.592,-124.143,170.305,46.949,159.015
C03228=1026.899,266.344,-124.113,170.301,46.950,159.015
C03229=1026.891,266.096,-124.083,170.297,46.952,159.015
C03230=1026.885,265.848,-124.054,170.293,46.954,159.015
C03231=1026.878,265.599,-124.024,170.289,46.956,159.015
C03232=1026.872,265.352,-123.994,170.285,46.958,159.014
C03233=1026.865,265.103,-123.963,170.281,46.959,159.014
C03234=1026.859,264.855,-123.934,170.277,46.961,159.014
C03235=1026.852,264.607,-123.904,170.274,46.963,159.014
C03236=1026.845,264.359,-123.875,170.269,46.965,159.014
C03237=1026.838,264.111,-123.845,170.265,46.966,159.014
C03238=1026.828,263.720,-123.798,170.260,46.969,159.014
C03239=1026.819,263.330,-123.751,170.253,46.972,159.014
C03240=1026.807,262.939,-123.704,170.248,46.975,159.014
C03241=1026.798,262.548,-123.658,170.241,46.978,159.013
C03242=1026.791,262.300,-123.628,170.237,46.980,159.013
C03243=1026.784,262.052,-123.599,170.234,46.981,159.013
C03244=1026.778,261.804,-123.569,170.230,46.983,159.013
C03245=1026.771,261.555,-123.539,170.226,46.985,159.013
C03246=1026.765,261.308,-123.509,170.223,46.987,159.013
C03247=1026.758,261.059,-123.480,170.218,46.989,159.013
C03248=1026.752,260.811,-123.450,170.214,46.991,159.013
C03249=1026.746,260.563,-123.421,170.210,46.993,159.013
C03250=1026.738,260.315,-123.392,170.207,46.995,159.013
C03251=1026.731,260.067,-123.362,170.203,46.997,159.013
C03252=1026.725,259.818,-123.333,170.200,46.999,159.013
C03253=1026.718,259.570,-123.304,170.195,47.001,159.013
C03254=1026.711,259.322,-123.274,170.191,47.003,159.013
C03255=1026.704,259.074,-123.245,170.188,47.005,159.013
C03256=1026.698,258.826,-123.216,170.184,47.007,159.013
C03257=1026.691,258.577,-123.187,170.180,47.009,159.013
C03258=1026.685,258.329,-123.158,170.176,47.011,159.013
C03259=1026.678,258.082,-123.129,170.172,47.013,159.012
C03260=1026.671,257.833,-123.099,170.169,47.015,159.013
C03261=1026.664,257.585,-123.070,170.165,47.017,159.012
C03262=1026.658,257.336,-123.041,170.162,47.019,159.013
C03263=1026.651,257.088,-123.012,170.158,47.021,159.012
C03264=1026.644,256.840,-122.983,170.153,47.023,159.012
C03265=1026.638,256.591,-122.954,170.150,47.025,159.012
C03266=1026.631,256.344,-122.924,170.146,47.027,159.012
C03267=1026.625,256.096,-122.895,170.143,47.030,159.012
C03268=1026.617,255.847,-122.866,170.139,47.031,159.012
C03269=1026.611,255.599,-122.837,170.135,47.034,159.012
C03270=1026.605,255.351,-122.808,170.132,47.035,159.012
C03271=1026.598,255.102,-122.779,170.127,47.038,159.012
C03272=1026.591,254.854,-122.750,170.123,47.040,159.012
C03273=1026.585,254.606,-122.721,170.120,47.042,159.012
C03274=1026.578,254.358,-122.692,170.116,47.044,159.012
C03275=1026.571,254.109,-122.663,170.113,47.046,159.012
C03276=1026.564,253.861,-122.634,170.109,47.048,159.012
C03277=1026.558,253.613,-122.605,170.106,47.050,159.012
C03278=1026.552,253.365,-122.576,170.102,47.052,159.012
C03279=1026.545,253.116,-122.547,170.097,47.055,159.012
C03280=1026.538,252.868,-122.518,170.094,47.057,159.012
C03281=1026.532,252.620,-122.489,170.090,47.059,159.012
C03282=1026.526,252.372,-122.460,170.087,47.061,159.012
C03283=1026.519,252.123,-122.431,170.083,47.063,159.012
C03284=1026.512,251.875,-122.402,170.080,47.065,159.012
C03285=1026.506,251.627,-122.373,170.076,47.067,159.012
C03286=1026.499,251.379,-122.344,170.072,47.069,159.012
C03287=1026.493,251.130,-122.316,170.069,47.072,159.012
C03288=1026.486,250.882,-122.287,170.065,47.073,159.012
C03289=1026.480,250.634,-122.258,170.061,47.076,159.012
C03290=1026.473,250.386,-122.229,170.057,47.078,159.012
C03291=1026.467,250.137,-122.200,170.054,47.080,159.012
C03292=1026.460,249.890,-122.172,170.050,47.082,159.012
C03293=1026.454,249.642,-122.143,170.046,47.084,159.012
C03294=1026.443,249.249,-122.098,170.041,47.088,159.012
C03295=1026.434,248.857,-122.052,170.035,47.092,159.012
C03296=1026.423,248.464,-122.007,170.030,47.094,159.012
C03297=1026.413,248.072,-121.961,170.023,47.098,159.012
C03298=1026.406,247.824,-121.932,170.020,47.101,159.013
C03299=1026.400,247.576,-121.904,170.016,47.102,159.012
C03300=1026.394,247.327,-121.875,170.013,47.105,159.013
C03301=1026.387,247.080,-121.846,170.009,47.107,159.013
C03302=1026.381,246.832,-121.817,170.006,47.109,159.013
C03303=1026.375,246.583,-121.789,170.002,47.111,159.013
C03304=1026.368,246.335,-121.760,169.999,47.114,159.013
C03305=1026.362,246.087,-121.731,169.995,47.115,159.013
C03306=1026.356,245.838,-121.703,169.992,47.118,159.013
C03307=1026.350,245.590,-121.674,169.988,47.120,159.013
C03308=1026.343,245.341,-121.646,169.985,47.122,159.013
C03309=1026.337,245.093,-121.617,169.981,47.124,159.013
C03310=1026.330,244.845,-121.588,169.978,47.127,159.013
C03311=1026.324,244.596,-121.560,169.974,47.129,159.013
C03312=1026.317,244.349,-121.531,169.971,47.131,159.013
C03313=1026.311,244.101,-121.502,169.967,47.133,159.013
C03314=1026.305,243.852,-121.474,169.964,47.135,159.013
C03315=1026.298,243.604,-121.446,169.960,47.138,159.013
C03316=1026.292,243.355,-121.418,169.956,47.140,159.013
C03317=1026.286,243.107,-121.390,169.952,47.143,159.013
C03318=1026.279,242.859,-121.361,169.949,47.145,159.013
C03319=1026.273,242.610,-121.333,169.945,47.148,159.013
C03320=1026.266,242.362,-121.304,169.942,47.150,159.013
C03321=1026.260,242.114,-121.276,169.938,47.152,159.013
C03322=1026.253,241.866,-121.248,169.935,47.155,159.014
C03323=1026.247,241.617,-121.219,169.931,47.156,159.013
C03324=1026.240,241.369,-121.192,169.928,47.159,159.013
C03325=1026.233,241.121,-121.163,169.924,47.161,159.014
C03326=1026.227,240.872,-121.135,169.921,47.164,159.014
C03327=1026.221,240.624,-121.107,169.918,47.166,159.014
C03328=1026.214,240.375,-121.078,169.914,47.168,159.014
C03329=1026.208,240.127,-121.050,169.911,47.171,159.014
C03330=1026.202,239.878,-121.022,169.907,47.173,159.014
C03331=1026.195,239.630,-120.993,169.904,47.175,159.014
C03332=1026.188,239.382,-120.966,169.900,47.178,159.014
C03333=1026.181,239.134,-120.938,169.896,47.181,159.014
C03334=1026.175,238.885,-120.910,169.893,47.184,159.014
C03335=1026.169,238.636,-120.882,169.889,47.186,159.014
C03336=1026.162,238.388,-120.854,169.886,47.188,159.015
C03337=1026.155,238.140,-120.826,169.882,47.191,159.015
C03338=1026.148,237.892,-120.798,169.879,47.193,159.015
C03339=1026.142,237.643,-120.770,169.876,47.195,159.015
C03340=1026.136,237.394,-120.742,169.872,47.198,159.015
C03341=1026.130,237.147,-120.715,169.869,47.201,159.015
C03342=1026.123,236.898,-120.687,169.866,47.203,159.015
C03343=1026.116,236.650,-120.659,169.862,47.206,159.015
C03344=1026.110,236.401,-120.631,169.859,47.208,159.015
C03345=1026.103,236.153,-120.604,169.855,47.210,159.015
C03346=1026.096,235.904,-120.576,169.852,47.213,159.016
C03347=1026.090,235.656,-120.548,169.848,47.216,159.016
C03348=1026.084,235.407,-120.520,169.844,47.219,159.016
C03349=1026.077,235.159,-120.492,169.841,47.221,159.016
C03350=1026.066,234.761,-120.447,169.836,47.225,159.016
C03351=1026.056,234.363,-120.403,169.830,47.229,159.016
C03352=1026.045,233.965,-120.359,169.825,47.233,159.016
C03353=1026.035,233.566,-120.314,169.819,47.238,159.017
C03354=1026.028,233.318,-120.286,169.816,47.240,159.017
C03355=1026.022,233.070,-120.259,169.812,47.243,159.017
C03356=1026.016,232.821,-120.232,169.809,47.245,159.017
C03357=1026.009,232.572,-120.204,169.806,47.248,159.017
C03358=1026.003,232.324,-120.176,169.802,47.250,159.017
C03359=1025.996,232.076,-120.149,169.799,47.253,159.017
C03360=1025.990,231.828,-120.121,169.796,47.256,159.018
C03361=1025.984,231.579,-120.093,169.792,47.258,159.018
C03362=1025.977,231.331,-120.065,169.789,47.261,159.018
C03363=1025.971,231.082,-120.038,169.785,47.263,159.018
C03364=1025.964,230.833,-120.011,169.782,47.266,159.018
C03365=1025.958,230.585,-119.983,169.779,47.268,159.018
C03366=1025.951,230.337,-119.955,169.776,47.271,159.018
C03367=1025.945,230.089,-119.928,169.772,47.274,159.018
C03368=1025.938,229.839,-119.901,169.769,47.276,159.019
C03369=1025.932,229.592,-119.873,169.766,47.279,159.019
C03370=1025.926,229.343,-119.846,169.762,47.282,159.019
C03371=1025.919,229.095,-119.818,169.759,47.285,159.019
C03372=1025.912,228.846,-119.791,169.756,47.287,159.019
C03373=1025.906,228.598,-119.764,169.752,47.289,159.019
C03374=1025.899,228.350,-119.736,169.749,47.293,159.019
C03375=1025.893,228.101,-119.709,169.745,47.295,159.019
C03376=1025.886,227.852,-119.682,169.742,47.298,159.020
C03377=1025.880,227.605,-119.654,169.738,47.301,159.020
C03378=1025.874,227.356,-119.627,169.735,47.304,159.020
C03379=1025.867,227.107,-119.599,169.732,47.306,159.020
C03380=1025.861,226.859,-119.573,169.729,47.309,159.020
C03381=1025.854,226.611,-119.546,169.725,47.312,159.020
C03382=1025.847,226.362,-119.518,169.722,47.315,159.021
C03383=1025.841,226.113,-119.491,169.719,47.318,159.021
C03384=1025.834,225.866,-119.464,169.715,47.320,159.021
C03385=1025.827,225.617,-119.437,169.712,47.323,159.021
C03386=1025.821,225.368,-119.409,169.709,47.325,159.021
C03387=1025.815,225.120,-119.383,169.706,47.328,159.022
C03388=1025.808,224.871,-119.356,169.703,47.332,159.022
C03389=1025.801,224.623,-119.329,169.699,47.334,159.022
C03390=1025.795,224.374,-119.302,169.696,47.337,159.022
C03391=1025.788,224.126,-119.275,169.693,47.339,159.022
C03392=1025.782,223.877,-119.248,169.689,47.342,159.023
C03393=1025.776,223.629,-119.220,169.685,47.346,159.023
C03394=1025.768,223.381,-119.194,169.682,47.348,159.023
C03395=1025.762,223.132,-119.167,169.679,47.351,159.023
C03396=1025.756,222.884,-119.140,169.676,47.354,159.023
C03397=1025.750,222.635,-119.113,169.672,47.357,159.023
C03398=1025.742,222.387,-119.086,169.669,47.360,159.024
C03399=1025.736,222.138,-119.059,169.666,47.363,159.024
C03400=1025.730,221.889,-119.032,169.663,47.365,159.024
C03401=1025.723,221.642,-119.005,169.659,47.368,159.024
C03402=1025.717,221.393,-118.978,169.656,47.371,159.024
C03403=1025.710,221.144,-118.951,169.653,47.374,159.024
C03404=1025.704,220.896,-118.924,169.650,47.377,159.025
C03405=1025.697,220.647,-118.897,169.647,47.380,159.025
C03406=1025.687,220.241,-118.853,169.641,47.384,159.025
C03407=1025.676,219.835,-118.809,169.636,47.389,159.026
C03408=1025.666,219.429,-118.766,169.630,47.394,159.026
C03409=1025.655,219.023,-118.722,169.626,47.399,159.026
C03410=1025.649,218.774,-118.695,169.622,47.401,159.026
C03411=1025.642,218.526,-118.668,169.619,47.404,159.027
C03412=1025.636,218.278,-118.642,169.616,47.407,159.027
C03413=1025.629,218.029,-118.615,169.613,47.410,159.027
C03414=1025.623,217.781,-118.588,169.609,47.414,159.027
C03415=1025.616,217.532,-118.562,169.606,47.417,159.028
C03416=1025.609,217.284,-118.536,169.603,47.420,159.028
C03417=1025.603,217.035,-118.509,169.600,47.423,159.028
C03418=1025.597,216.787,-118.483,169.596,47.426,159.028
C03419=1025.590,216.538,-118.456,169.593,47.428,159.028
C03420=1025.583,216.289,-118.429,169.590,47.431,159.029
C03421=1025.576,216.041,-118.403,169.587,47.434,159.029
C03422=1025.570,215.792,-118.376,169.584,47.437,159.029
C03423=1025.563,215.544,-118.350,169.581,47.441,159.029
C03424=1025.557,215.295,-118.323,169.577,47.444,159.030
C03425=1025.550,215.047,-118.297,169.574,47.447,159.030
C03426=1025.543,214.798,-118.270,169.571,47.450,159.030
C03427=1025.538,214.550,-118.243,169.568,47.453,159.030
C03428=1025.530,214.301,-118.217,169.565,47.456,159.031
C03429=1025.525,214.053,-118.190,169.562,47.459,159.031
C03430=1025.518,213.804,-118.165,169.559,47.462,159.031
C03431=1025.511,213.556,-118.139,169.556,47.465,159.031
C03432=1025.506,213.307,-118.112,169.553,47.468,159.032
C03433=1025.499,213.058,-118.086,169.549,47.471,159.032
C03434=1025.493,212.810,-118.059,169.546,47.474,159.032
C03435=1025.486,212.561,-118.033,169.542,47.478,159.032
C03436=1025.479,212.313,-118.006,169.539,47.481,159.032
C03437=1025.473,212.064,-117.979,169.536,47.484,159.033
C03438=1025.466,211.816,-117.953,169.533,47.487,159.033
C03439=1025.459,211.567,-117.927,169.530,47.490,159.033
C03440=1025.453,211.319,-117.900,169.527,47.493,159.033
C03441=1025.447,211.071,-117.874,169.523,47.496,159.034
C03442=1025.441,210.821,-117.848,169.520,47.499,159.034
C03443=1025.434,210.573,-117.822,169.517,47.502,159.034
C03444=1025.427,210.325,-117.796,169.514,47.505,159.034
C03445=1025.421,210.077,-117.769,169.511,47.508,159.035
C03446=1025.415,209.828,-117.743,169.508,47.511,159.035
C03447=1025.408,209.579,-117.717,169.505,47.514,159.035
C03448=1025.402,209.331,-117.691,169.502,47.518,159.035
C03449=1025.394,209.082,-117.665,169.499,47.521,159.036
C03450=1025.388,208.834,-117.639,169.496,47.524,159.036
C03451=1025.382,208.585,-117.613,169.493,47.527,159.036
C03452=1025.375,208.336,-117.586,169.490,47.531,159.037
C03453=1025.369,208.088,-117.560,169.486,47.534,159.037
C03454=1025.362,207.839,-117.534,169.483,47.537,159.037
C03455=1025.355,207.591,-117.508,169.480,47.540,159.037
C03456=1025.349,207.343,-117.482,169.477,47.543,159.038
C03457=1025.343,207.093,-117.456,169.474,47.547,159.038
C03458=1025.336,206.845,-117.430,169.471,47.550,159.038
C03459=1025.330,206.597,-117.404,169.468,47.553,159.039
C03460=1025.323,206.348,-117.378,169.465,47.556,159.039
C03461=1025.317,206.100,-117.352,169.461,47.560,159.039
C03462=1025.306,205.696,-117.310,169.457,47.565,159.039
C03463=1025.295,205.292,-117.268,169.451,47.571,159.040
C03464=1025.285,204.890,-117.226,169.447,47.576,159.040
C03465=1025.274,204.487,-117.185,169.442,47.581,159.041
C03466=1025.250,203.453,-117.084,169.042,47.480,158.967
C03467=1025.244,203.204,-117.059,169.038,47.484,158.967
C03468=1025.239,202.955,-117.035,169.035,47.488,158.968
C03469=1025.233,202.706,-117.010,169.030,47.492,158.968
C03470=1025.227,202.458,-116.985,169.026,47.496,158.968
C03471=1025.221,202.209,-116.961,169.022,47.500,158.969
C03472=1025.215,201.960,-116.937,169.018,47.504,158.969
C03473=1025.210,201.712,-116.913,169.013,47.508,158.969
C03474=1025.204,201.462,-116.888,169.010,47.513,158.970
C03475=1025.198,201.214,-116.864,169.006,47.517,158.970
C03476=1025.193,200.966,-116.840,169.002,47.521,158.970
C03477=1025.187,200.716,-116.816,168.998,47.525,158.971
C03478=1025.182,200.468,-116.791,168.994,47.529,158.971
C03479=1025.176,200.218,-116.767,168.990,47.533,158.971
C03480=1025.170,199.970,-116.743,168.986,47.537,158.972
C03481=1025.164,199.722,-116.719,168.982,47.541,158.972
C03482=1025.158,199.473,-116.695,168.978,47.546,158.972
C03483=1025.153,199.223,-116.671,168.973,47.550,158.973
C03484=1025.146,198.974,-116.647,168.970,47.554,158.973
C03485=1025.141,198.726,-116.623,168.966,47.559,158.973
C03486=1025.135,198.478,-116.599,168.962,47.563,158.974
C03487=1025.128,198.229,-116.575,168.957,47.568,158.974
C03488=1025.123,197.979,-116.552,168.954,47.572,158.974
C03489=1025.117,197.731,-116.528,168.950,47.576,158.975
C03490=1025.111,197.482,-116.503,168.946,47.580,158.975
C03491=1025.105,197.234,-116.480,168.942,47.584,158.975
C03492=1025.099,196.985,-116.457,168.938,47.589,158.976
C03493=1025.093,196.735,-116.432,168.934,47.593,158.976
C03494=1025.087,196.487,-116.408,168.930,47.597,158.976
C03495=1025.082,196.238,-116.384,168.926,47.601,158.977
C03496=1025.076,195.990,-116.361,168.923,47.606,158.977
C03497=1025.070,195.740,-116.337,168.918,47.610,158.978
C03498=1025.064,195.492,-116.313,168.914,47.614,158.978
C03499=1025.059,195.243,-116.290,168.911,47.619,158.978
C03500=1025.053,194.995,-116.266,168.907,47.623,158.979
C03501=1025.047,194.745,-116.242,168.903,47.627,158.979
C03502=1025.042,194.496,-116.218,168.899,47.632,158.980
C03503=1025.036,194.248,-116.195,168.895,47.636,158.980
C03504=1025.030,193.999,-116.172,168.891,47.640,158.980
C03505=1025.024,193.750,-116.147,168.887,47.645,158.981
C03506=1025.018,193.502,-116.123,168.883,47.649,158.981
C03507=1025.013,193.252,-116.100,168.880,47.653,158.981
C03508=1025.007,193.004,-116.076,168.876,47.658,158.982
C03509=1025.001,192.755,-116.053,168.872,47.662,158.982
C03510=1024.995,192.506,-116.029,168.867,47.666,158.982
C03511=1024.990,192.257,-116.006,168.864,47.671,158.983
C03512=1024.984,192.009,-115.982,168.860,47.675,158.983
C03513=1024.979,191.760,-115.958,168.856,47.679,158.983
C03514=1024.973,191.511,-115.935,168.853,47.684,158.984
C03515=1024.967,191.261,-115.911,168.849,47.688,158.984
C03516=1024.961,191.013,-115.887,168.845,47.692,158.985
C03517=1024.955,190.764,-115.864,168.842,47.696,158.985
C03518=1024.950,190.516,-115.840,168.838,47.700,158.985
C03519=1024.944,190.267,-115.817,168.834,47.705,158.986
C03520=1024.939,190.018,-115.793,168.829,47.710,158.986
C03521=1024.933,189.769,-115.770,168.825,47.714,158.986
C03522=1024.927,189.521,-115.746,168.822,47.718,158.987
C03523=1024.922,189.271,-115.722,168.818,47.722,158.987
C03524=1024.916,189.022,-115.699,168.814,47.726,158.988
C03525=1024.910,188.774,-115.676,168.811,47.731,158.988
C03526=1024.905,188.525,-115.652,168.807,47.735,158.988
C03527=1024.898,188.243,-115.626,168.802,47.740,158.989
C03528=1024.892,187.960,-115.599,168.799,47.745,158.989
C03529=1024.886,187.677,-115.572,168.794,47.750,158.990
C03530=1024.879,187.395,-115.546,168.790,47.755,158.990
C03531=1024.874,187.146,-115.523,168.786,47.759,158.990
C03532=1024.868,186.898,-115.499,168.783,47.764,158.991
C03533=1024.863,186.649,-115.476,168.779,47.768,158.991
C03534=1024.858,186.400,-115.452,168.775,47.772,158.991
C03535=1024.852,186.151,-115.429,168.771,47.777,158.992
C03536=1024.846,185.902,-115.406,168.768,47.781,158.992
C03537=1024.841,185.653,-115.382,168.764,47.785,158.993
C03538=1024.835,185.405,-115.359,168.760,47.789,158.993
C03539=1024.829,185.156,-115.336,168.756,47.793,158.993
C03540=1024.824,184.907,-115.312,168.753,47.798,158.994
C03541=1024.818,184.658,-115.289,168.749,47.802,158.994
C03542=1024.813,184.409,-115.266,168.746,47.807,158.995
C03543=1024.807,184.160,-115.242,168.742,47.811,158.995
C03544=1024.802,183.912,-115.219,168.738,47.815,158.995
C03545=1024.796,183.663,-115.196,168.734,47.820,158.996
C03546=1024.791,183.413,-115.172,168.731,47.824,158.996
C03547=1024.785,183.165,-115.149,168.727,47.829,158.997
C03548=1024.780,182.915,-115.126,168.724,47.832,158.997
C03549=1024.774,182.667,-115.102,168.720,47.836,158.997
C03550=1024.768,182.418,-115.079,168.717,47.841,158.998
C03551=1024.763,182.169,-115.057,168.712,47.846,158.998
C03552=1024.757,181.920,-115.034,168.709,47.850,158.999
C03553=1024.751,181.671,-115.012,168.705,47.855,158.999
C03554=1024.745,181.422,-114.989,168.702,47.860,159.000
C03555=1024.739,181.173,-114.966,168.698,47.865,159.000
C03556=1024.734,180.925,-114.943,168.694,47.869,159.000
C03557=1024.727,180.676,-114.921,168.691,47.873,159.001
C03558=1024.721,180.427,-114.898,168.687,47.878,159.001
C03559=1024.716,180.178,-114.875,168.684,47.883,159.002
C03560=1024.710,179.929,-114.853,168.680,47.887,159.002
C03561=1024.704,179.680,-114.830,168.677,47.892,159.003
C03562=1024.698,179.431,-114.807,168.673,47.896,159.003
C03563=1024.692,179.182,-114.784,168.670,47.901,159.004
C03564=1024.687,178.933,-114.762,168.666,47.905,159.004
C03565=1024.680,178.684,-114.740,168.662,47.910,159.004
C03566=1024.675,178.435,-114.717,168.659,47.915,159.005
C03567=1024.669,178.186,-114.694,168.655,47.919,159.005
C03568=1024.663,177.937,-114.672,168.651,47.924,159.006
C03569=1024.657,177.688,-114.649,168.648,47.928,159.006
C03570=1024.652,177.440,-114.627,168.644,47.933,159.007
C03571=1024.646,177.191,-114.604,168.641,47.938,159.007
C03572=1024.640,176.942,-114.582,168.637,47.942,159.007
C03573=1024.634,176.693,-114.559,168.634,47.947,159.008
C03574=1024.629,176.444,-114.536,168.630,47.951,159.008
C03575=1024.623,176.195,-114.514,168.627,47.956,159.009
